(* IEC 61131-3 sources: RL_MAR/experiments/results/ablation/Ablation_antlr_only_deepseek-ai_DeepSeek-V3.2_20260611_164353 (part 2) *)

(* ---- med_34.st ---- *)
FUNCTION_BLOCK CoffeeMachineControl
VAR_INPUT
    StartButton : BOOL;
    ElapsedTime : DINT; (* Time elapsed since the start of the current process, in milliseconds *)
END_VAR

VAR_OUTPUT
    WaterHeating : BOOL;
    GrinderRunning : BOOL;
    Brewing : BOOL;
    GrinderFinished : BOOL;
    WaterHeated : BOOL;
    CoffeeReady : BOOL;
END_VAR

VAR
    (* Timing constants *)
    WaterHeatingDuration : DINT := 30000; (* 30 seconds in milliseconds *)
    GrinderDuration : DINT := 15000; (* 15 seconds in milliseconds *)
    BrewingDuration : DINT := 60000; (* 60 seconds in milliseconds *)

    (* State management *)
    CurrentState : INT := 0; (* 0: Idle, 1: Heating, 2: Grinding, 3: Brewing *)
    ProcessStartTime : DINT := 0;

    (* Internal flags for process completion *)
    WaterHeatingDone : BOOL := FALSE;
    GrinderDone : BOOL := FALSE;
    BrewingDone : BOOL := FALSE;
END_VAR

(* Main state machine logic *)
IF NOT StartButton THEN
    (* Reset everything when start button is not pressed *)
    CurrentState := 0;
    ProcessStartTime := 0;
    WaterHeatingDone := FALSE;
    GrinderDone := FALSE;
    BrewingDone := FALSE;

    WaterHeating := FALSE;
    GrinderRunning := FALSE;
    Brewing := FALSE;
    WaterHeated := FALSE;
    GrinderFinished := FALSE;
    CoffeeReady := FALSE;
ELSE
    (* Process state machine *)
    CASE CurrentState OF
        0: (* Idle - waiting for start *)
            IF StartButton AND NOT WaterHeatingDone THEN
                CurrentState := 1;
                ProcessStartTime := ElapsedTime;
                WaterHeating := TRUE;
            END_IF;

        1: (* Water Heating *)
            WaterHeating := TRUE;
            WaterHeated := FALSE;

            IF (ElapsedTime - ProcessStartTime) >= WaterHeatingDuration THEN
                WaterHeating := FALSE;
                WaterHeatingDone := TRUE;
                WaterHeated := TRUE;
                CurrentState := 2;
                ProcessStartTime := ElapsedTime;
            END_IF;

        2: (* Grinding *)
            IF WaterHeatingDone AND NOT GrinderDone THEN
                GrinderRunning := TRUE;
                GrinderFinished := FALSE;

                IF (ElapsedTime - ProcessStartTime) >= GrinderDuration THEN
                    GrinderRunning := FALSE;
                    GrinderDone := TRUE;
                    GrinderFinished := TRUE;
                    CurrentState := 3;
                    ProcessStartTime := ElapsedTime;
                END_IF;
            END_IF;

        3: (* Brewing *)
            IF GrinderDone AND NOT BrewingDone THEN
                Brewing := TRUE;
                CoffeeReady := FALSE;

                IF (ElapsedTime - ProcessStartTime) >= BrewingDuration THEN
                    Brewing := FALSE;
                    BrewingDone := TRUE;
                    CoffeeReady := TRUE;
                    (* Stay in state 3 until reset *)
                END_IF;
            END_IF;

    END_CASE;
END_IF;

END_FUNCTION_BLOCK;

(* ---- med_35.st ---- *)
FUNCTION_BLOCK FB_SimpleCalculation
VAR_INPUT
    INPUT_VAR1 : INT := 2;
    VAR2 : INT := 0;
END_VAR

VAR_OUTPUT
    OUTPUT_VAR1 : INT;
    OUTPUT_VAR2 : INT;
END_VAR

VAR
    i : INT; // Loop counter for multiplication
    j : INT; // Loop counter for increment
END_VAR

// Main logic
OUTPUT_VAR1 := INPUT_VAR1; // Initial assignment as per requirements

// First loop: Multiply OUTPUT_VAR1 by 2 for exactly 5 iterations
FOR i := 1 TO 5 DO
    OUTPUT_VAR1 := OUTPUT_VAR1 * 2;
END_FOR;

OUTPUT_VAR2 := VAR2; // Initial assignment as per requirements

// Second loop: Increment OUTPUT_VAR2 by 1 for exactly 5 iterations
FOR j := 1 TO 5 DO
    OUTPUT_VAR2 := OUTPUT_VAR2 + 1;
END_FOR;

END_FUNCTION_BLOCK

(* ---- med_36.st ---- *)
(*
    FUNCTION_BLOCK: FB_ExpandedPoint
    Description: Processes input values and assigns specific constant values to outputs.
    Inputs:
        INPUT_VAR2   : INT - Directly passed to OUTPUT_VAR2.
        INPUT_VAR1_X : INT - Unused input.
        INPUT_VAR1_Y : INT - Unused input.
        INPUT_VAR3_X : INT := 1 - Unused input with default value.
        INPUT_VAR3_Y : INT := 2 - Unused input with default value.
    Outputs:
        OUTPUT_VAR2   : INT - Assigned the value of INPUT_VAR2.
        OUTPUT_VAR1_X : INT - Assigned constant value 1.
        OUTPUT_VAR1_Y : INT - Assigned constant value 2.
        OUTPUT_VAR3_X : INT - Assigned constant value 100.
        OUTPUT_VAR3_Y : INT - Assigned constant value -7000.
    Logic: Stateless, deterministic assignments executed every cycle.
*)

FUNCTION_BLOCK FB_ExpandedPoint
VAR_INPUT
    INPUT_VAR2 : INT;
    INPUT_VAR1_X : INT;
    INPUT_VAR1_Y : INT;
    INPUT_VAR3_X : INT := 1;
    INPUT_VAR3_Y : INT := 2;
END_VAR

VAR_OUTPUT
    OUTPUT_VAR2 : INT;
    OUTPUT_VAR1_X : INT;
    OUTPUT_VAR1_Y : INT;
    OUTPUT_VAR3_X : INT;
    OUTPUT_VAR3_Y : INT;
END_VAR

// No internal variables required for this stateless function block.

// --- Main Execution Logic ---
// Executes unconditionally every cycle.
OUTPUT_VAR2 := INPUT_VAR2;
OUTPUT_VAR1_X := 1;
OUTPUT_VAR1_Y := 2;
OUTPUT_VAR3_X := 100;
OUTPUT_VAR3_Y := -7000;

END_FUNCTION_BLOCK

(* ---- med_37.st ---- *)
FUNCTION_BLOCK FB_RealValueAdjuster
VAR_INPUT
    x_in : REAL;
END_VAR

VAR_OUTPUT
    x_out : REAL;
END_VAR

VAR
    x : REAL;
    int_val : INT;
END_VAR

(* Initialize the working variable with the input *)
x := x_in;

(* Process the input based on the defined rules *)
(* Rule 1 & 2: Add 1.0 if input is exactly 0.0 OR if input is not 0.0 *)
(* Since both conditions are mutually exclusive and cover all possibilities, this is an unconditional addition of 1.0 *)
x := x + 1.0;

(* Rule 3: Equality and inequality check - already satisfied by the unconditional addition above *)
(* No additional conditional logic required as the operation is already performed *)

(* Rule 4: Convert the original real input to an integer and, if the integer conversion is not zero, add 1.0 to the original real input *)
(* Note: The requirement specifies using the original real input (x_in) for this check *)
int_val := REAL_TO_INT(x_in);
IF int_val <> 0 THEN
    x := x + 1.0;
END_IF;

(* Assign the final result to the output *)
x_out := x;

END_FUNCTION_BLOCK

(* ---- med_38.st ---- *)
FUNCTION_BLOCK SolarPanelTracking
VAR_INPUT
    SolarIntensity : REAL;      (* Input: Solar intensity in percentage *)
    CurrentTime : TIME;         (* Input: Current time of day *)
END_VAR

VAR_OUTPUT
    PanelAngle : REAL := 0.0;   (* Output: Panel angle in degrees *)
END_VAR

VAR
    SunriseTime : TIME := T#6H;    (* Sunrise time set to 6 AM *)
    SunsetTime : TIME := T#18H;    (* Sunset time set to 6 PM *)
    NoonTime : TIME := T#12H;      (* Noon time set to 12 PM *)
    MorningAngle : REAL := 30.0;   (* Angle during morning *)
    NoonAngle : REAL := 60.0;      (* Angle during noon *)
    EveningAngle : REAL := 30.0;   (* Angle during evening *)
    State : INT := 0;
    NextState : INT := 0;
END_VAR

CASE State OF
    0: (* INIT *)
        PanelAngle := 0.0;
        SunriseTime := T#6H;
        SunsetTime := T#18H;
        NoonTime := T#12H;
        MorningAngle := 30.0;
        NoonAngle := 60.0;
        EveningAngle := 30.0;
        NextState := 1;

    1: (* CHECK_TIME *)
        IF (CurrentTime < SunriseTime) OR (CurrentTime >= SunsetTime) THEN
            NextState := 2;  (* NIGHTTIME *)
        ELSIF (CurrentTime >= SunriseTime) AND (CurrentTime < NoonTime) THEN
            NextState := 3;  (* MORNING *)
        ELSIF (CurrentTime >= NoonTime) AND (CurrentTime < SunsetTime) THEN
            NextState := 4;  (* AFTERNOON *)
        ELSE
            NextState := 1;  (* Stay in CHECK_TIME *)
        END_IF;

    2: (* NIGHTTIME *)
        PanelAngle := 0.0;
        NextState := 1;

    3: (* MORNING *)
        IF SolarIntensity >= 90.0 THEN
            PanelAngle := NoonAngle;
        ELSE
            PanelAngle := MorningAngle;
        END_IF;

        (* Clamp angle to 0-90 degrees *)
        IF PanelAngle < 0.0 THEN
            PanelAngle := 0.0;
        ELSIF PanelAngle > 90.0 THEN
            PanelAngle := 90.0;
        END_IF;
        NextState := 1;

    4: (* AFTERNOON *)
        IF SolarIntensity >= 90.0 THEN
            PanelAngle := NoonAngle;
        ELSE
            PanelAngle := EveningAngle;
        END_IF;

        (* Clamp angle to 0-90 degrees *)
        IF PanelAngle < 0.0 THEN
            PanelAngle := 0.0;
        ELSIF PanelAngle > 90.0 THEN
            PanelAngle := 90.0;
        END_IF;
        NextState := 1;

END_CASE;

State := NextState;

END_FUNCTION_BLOCK

(* ---- med_39.st ---- *)
FUNCTION_BLOCK WindTurbineControl
VAR_INPUT
    WindSpeedSensor : REAL; (* Input for measuring wind speed *)
    GeneratorSpeedSensor : REAL; (* Input for measuring generator speed *)
END_VAR

VAR_OUTPUT
    BladePitch : INT; (* Output for blade pitch control (degrees) *)
    GeneratorSpeed : REAL; (* Output for generator speed control (RPM) *)
END_VAR

VAR
    (* No internal variables needed for this simple logic *)
END_VAR

(* Main control logic *)
IF WindSpeedSensor <= 3.0 THEN
    (* Low wind speed category *)
    BladePitch := -5;
    GeneratorSpeed := 500.0;
ELSIF (WindSpeedSensor > 3.0) AND (WindSpeedSensor <= 5.0) THEN
    (* Moderate wind speed category *)
    BladePitch := 0;
    GeneratorSpeed := 800.0;
ELSE
    (* High wind speed category (WindSpeedSensor > 5.0) *)
    BladePitch := 5;
    GeneratorSpeed := 1000.0;
END_IF;

END_FUNCTION_BLOCK

(* ---- med_40.st ---- *)
FUNCTION_BLOCK RockClimbingWallControl
VAR_INPUT
    UserWeightSensor : REAL; (* Input for measuring the user's weight *)
    WallDifficultyLevel : INT; (* Input for setting the wall's initial difficulty level *)
    WallHeight : REAL; (* Input for setting the wall's height *)
    RouteSelector : INT; (* Input for selecting a climbing route *)
END_VAR
VAR_OUTPUT
    ClimbingMotorSpeed : REAL; (* Output for controlling the climbing wall motor speed *)
    WallLights : BOOL; (* Output for controlling wall lighting *)
END_VAR
VAR
    InternalWeightThreshold : REAL := 60.0;
    InternalHeightThreshold : REAL := 5.0;
    InternalRouteLevel : INT;
    InternalMotorSpeedAdjust : REAL;
    InternalLightCondition : BOOL;
END_VAR

(* Route-based difficulty level assignment *)
CASE RouteSelector OF
    1: InternalRouteLevel := 1;
    2: InternalRouteLevel := 2;
    3: InternalRouteLevel := 3;
ELSE
    InternalRouteLevel := WallDifficultyLevel; (* Fallback to initial difficulty level *)
END_CASE;

(* Motor speed adjustment based on user weight *)
IF UserWeightSensor > InternalWeightThreshold THEN
    InternalMotorSpeedAdjust := 1.0;
ELSE
    InternalMotorSpeedAdjust := 0.8;
END_IF;

(* Wall lighting control based on wall height *)
IF WallHeight > InternalHeightThreshold THEN
    InternalLightCondition := TRUE;
ELSE
    InternalLightCondition := FALSE;
END_IF;

(* Assign final output values *)
ClimbingMotorSpeed := InternalMotorSpeedAdjust;
WallLights := InternalLightCondition;

END_FUNCTION_BLOCK

(* ---- med_41.st ---- *)
FUNCTION_BLOCK FishTankControl
VAR_INPUT
    OxygenLevel : REAL; (* Input for oxygen level in the tank *)
    WaterTemperature : REAL; (* Input for water temperature *)
    FeedingTime : TIME; (* Time for scheduled feeding *)
    CurrentTime : TIME; (* Current system time *)
END_VAR
VAR_OUTPUT
    OxygenValve : BOOL; (* Output to control oxygen supply *)
    Heater : BOOL; (* Output to control the heater *)
    Feeder : BOOL; (* Output to control the fish feeder *)
END_VAR
VAR
    (* No internal variables required for basic threshold logic *)
END_VAR

(* Control logic for Oxygen Valve *)
IF OxygenLevel < 5.0 THEN
    OxygenValve := TRUE;
ELSE
    OxygenValve := FALSE;
END_IF;

(* Control logic for Heater *)
IF WaterTemperature < 25.0 THEN
    Heater := TRUE;
ELSE
    Heater := FALSE;
END_IF;

(* Control logic for Feeder *)
IF CurrentTime >= FeedingTime THEN
    Feeder := TRUE;
ELSE
    Feeder := FALSE;
END_IF;

END_FUNCTION_BLOCK

(* ---- med_42.st ---- *)
FUNCTION_BLOCK RetractableRoofControl
VAR_INPUT
    RainSensor : BOOL; (* TRUE = rain detected, FALSE = no rain *)
    WindSensor : BOOL; (* TRUE = wind detected, FALSE = no wind *)
    TemperatureSensor : REAL; (* Current temperature in degrees Celsius *)
END_VAR

VAR_OUTPUT
    RoofMotor : BOOL; (* TRUE = motor active (close/partially close), FALSE = motor inactive (open/fully closed) *)
END_VAR

VAR
    (* No internal variables required for this logic *)
END_VAR

(*
    Control Logic for Motorized Retractable Roof:
    1. Rain AND Wind: Close completely (RoofMotor = FALSE)
    2. Rain AND NOT Wind: Partially close (RoofMotor = TRUE)
    3. NOT Rain AND Temperature < 20.0°C: Close slightly (RoofMotor = TRUE)
    4. NOT Rain AND Temperature >= 20.0°C: Open fully (RoofMotor = FALSE)

    Priority is implicit in the IF-ELSIF structure.
*)

BEGIN
    IF RainSensor AND WindSensor THEN
        RoofMotor := FALSE; (* Close completely *)
    ELSIF RainSensor AND NOT WindSensor THEN
        RoofMotor := TRUE; (* Partially close *)
    ELSIF NOT RainSensor AND TemperatureSensor < 20.0 THEN
        RoofMotor := TRUE; (* Close slightly *)
    ELSIF NOT RainSensor AND TemperatureSensor >= 20.0 THEN
        RoofMotor := FALSE; (* Open fully *)
    ELSE
        (* Fallback/default case - maintain current state *)
        RoofMotor := RoofMotor;
    END_IF;
END_FUNCTION_BLOCK

(* ---- med_43.st ---- *)
FUNCTION_BLOCK SandwichMaker
VAR_INPUT
    BreadFeeder : BOOL; (* Input: Detects the presence of bread slices *)
    Ingredient1 : BOOL; (* Input: Detects the presence of Ingredient 1 (e.g., cheese) *)
    Ingredient2 : BOOL; (* Input: Detects the presence of Ingredient 2 (e.g., lettuce) *)
    Ingredient3 : BOOL; (* Input: Detects the presence of Ingredient 3 (e.g., tomatoes) *)
    Condiment1 : BOOL; (* Input: Detects the presence of Condiment 1 (e.g., mayo) *)
    Condiment2 : BOOL; (* Input: Detects the presence of Condiment 2 (e.g., mustard) *)
END_VAR
VAR_OUTPUT
    ConveyorMotor : BOOL; (* Output: Controls the conveyor belt motor *)
    AssembleMotor : BOOL; (* Output: Controls the sandwich assembly motor *)
END_VAR
VAR
    SliceCount : INT := 0; (* Counter for bread slices *)
    PrevBreadState : BOOL := FALSE; (* Previous state for edge detection *)
    AllIngredientsPresent : BOOL := FALSE; (* Combined ingredient condition *)
END_VAR

(* Edge detection for bread slice counting *)
IF BreadFeeder AND NOT PrevBreadState THEN
    SliceCount := SliceCount + 1;
END_IF;

(* Update previous state for next scan cycle *)
PrevBreadState := BreadFeeder;

(* Conveyor motor control: Run when bread is detected *)
ConveyorMotor := BreadFeeder;

(* Check if all ingredients and condiments are present *)
AllIngredientsPresent := Ingredient1 AND Ingredient2 AND Ingredient3 AND Condiment1 AND Condiment2;

(* Assembly motor control: Activate only when all conditions are met *)
AssembleMotor := (SliceCount >= 2) AND AllIngredientsPresent;

(* Reset slice counter after successful assembly *)
IF AssembleMotor THEN
    SliceCount := SliceCount - 2;
END_IF;

END_FUNCTION_BLOCK

(* ---- med_44.st ---- *)
(*
FUNCTION_BLOCK: DroneChargingStation
DESCRIPTION: Manages charging and deployment for three drones based on battery levels.
LOGIC: Implements a state machine with three states (Idle, Charging, Deployed).
       - Idle: Checks for drones with battery < 20% and starts charging the first one found.
                If no drones need charging and all batteries >= 20%, allows deployment.
       - Charging: Charges a specific drone for the configured ChargingTime.
       - Deployed: Monitors battery levels and recalls (returns to Idle) if any battery falls below 10%.
*)

FUNCTION_BLOCK DroneChargingStation
VAR_INPUT
    Drone1BatteryLevel : INT := 0; (* Battery level of Drone 1 (0-100%) *)
    Drone2BatteryLevel : INT := 0; (* Battery level of Drone 2 (0-100%) *)
    Drone3BatteryLevel : INT := 0; (* Battery level of Drone 3 (0-100%) *)
    ChargingTime : TIME := T#30s;  (* Required charging duration *)
END_VAR
VAR_OUTPUT
    Drone1Status : BOOL := FALSE;        (* TRUE if Drone 1 is charging *)
    Drone2Status : BOOL := FALSE;        (* TRUE if Drone 2 is charging *)
    Drone3Status : BOOL := FALSE;        (* TRUE if Drone 3 is charging *)
    ChargingStationStatus : BOOL := FALSE; (* TRUE if station is charging a drone *)
    DroneDeployed : BOOL := FALSE;       (* TRUE if a drone is deployed *)
END_VAR
VAR
    (* State Management *)
    CurrentState : INT := 0; (* 0: Idle, 1: Charging, 2: Deployed *)
    ChargingDrone : INT := 0; (* 0: None, 1: Drone1, 2: Drone2, 3: Drone3 *)
    TimeRemaining : TIME;
END_VAR

(* Main State Machine *)
CASE CurrentState OF
    0: (* IDLE STATE *)
        (* Reset charging outputs *)
        Drone1Status := FALSE;
        Drone2Status := FALSE;
        Drone3Status := FALSE;
        ChargingStationStatus := FALSE;
        DroneDeployed := FALSE;
        ChargingDrone := 0;

        (* Check for drones needing charge (priority: Drone1 > Drone2 > Drone3) *)
        IF Drone1BatteryLevel < 20 THEN
            ChargingDrone := 1;
            TimeRemaining := ChargingTime;
            CurrentState := 1;
        ELSIF Drone2BatteryLevel < 20 THEN
            ChargingDrone := 2;
            TimeRemaining := ChargingTime;
            CurrentState := 1;
        ELSIF Drone3BatteryLevel < 20 THEN
            ChargingDrone := 3;
            TimeRemaining := ChargingTime;
            CurrentState := 1;
        ELSE
            (* No drones need charging. Check if deployment is possible. *)
            (* Deployment allowed only if all batteries are at least 20% *)
            IF (Drone1BatteryLevel >= 20) AND (Drone2BatteryLevel >= 20) AND (Drone3BatteryLevel >= 20) THEN
                CurrentState := 2;
            ELSE
                CurrentState := 0;
            END_IF;
        END_IF;

    1: (* CHARGING STATE *)
        (* Set station status and the specific drone's charging status *)
        ChargingStationStatus := TRUE;
        CASE ChargingDrone OF
            1: Drone1Status := TRUE;
            2: Drone2Status := TRUE;
            3: Drone3Status := TRUE;
        END_CASE;

        (* Decrement the charging timer *)
        TimeRemaining := TimeRemaining - T#1ms;

        (* Check if charging is complete *)
        IF TimeRemaining <= T#0ms THEN
            (* Charging complete, return to Idle state *)
            CurrentState := 0;
        ELSE
            CurrentState := 1;
        END_IF;

    2: (* DEPLOYED STATE *)
        (* A drone is deployed. Station is not in use for charging. *)
        DroneDeployed := TRUE;
        ChargingStationStatus := FALSE;
        Drone1Status := FALSE;
        Drone2Status := FALSE;
        Drone3Status := FALSE;

        (* Recall condition: If ANY drone's battery falls below 10%, return to Idle *)
        IF (Drone1BatteryLevel < 10) OR (Drone2BatteryLevel < 10) OR (Drone3BatteryLevel < 10) THEN
            DroneDeployed := FALSE;
            CurrentState := 0;
        ELSE
            CurrentState := 2;
        END_IF;

END_CASE;

END_FUNCTION_BLOCK

(* ---- med_45.st ---- *)
FUNCTION_BLOCK AutomatedSmoothieMaker
VAR_INPUT
    BananaAvailable : BOOL;
    BerryMixAvailable : BOOL;
    SpinachAvailable : BOOL;
    YogurtAvailable : BOOL;
    CustomerPreference : INT;
END_VAR

VAR_OUTPUT
    BlenderMotor : BOOL;
    Dispenser : BOOL;
END_VAR

VAR
    RecipeValid : BOOL;
    IngredientsAvailable : BOOL;
END_VAR

(* Initialize internal variables *)
RecipeValid := FALSE;
IngredientsAvailable := FALSE;

(* Validate customer preference and check ingredient availability *)
CASE CustomerPreference OF
    1: (* Recipe 1: Banana, Berry Mix, Yogurt *)
        RecipeValid := TRUE;
        IngredientsAvailable := BananaAvailable AND BerryMixAvailable AND YogurtAvailable;
    2: (* Recipe 2: Berry Mix, Spinach, Yogurt *)
        RecipeValid := TRUE;
        IngredientsAvailable := BerryMixAvailable AND SpinachAvailable AND YogurtAvailable;
    3: (* Recipe 3: Banana, Spinach, Yogurt *)
        RecipeValid := TRUE;
        IngredientsAvailable := BananaAvailable AND SpinachAvailable AND YogurtAvailable;
    ELSE
        RecipeValid := FALSE;
        IngredientsAvailable := FALSE;
END_CASE;

(* Control outputs based on validation and availability *)
IF RecipeValid AND IngredientsAvailable THEN
    BlenderMotor := TRUE;
    Dispenser := TRUE;
ELSE
    BlenderMotor := FALSE;
    Dispenser := FALSE;
END_IF;

END_FUNCTION_BLOCK

(* ---- med_46.st ---- *)
FUNCTION_BLOCK PrecisionEngravingMachine
VAR_INPUT
    DesignSelection : INT;
END_VAR

VAR_OUTPUT
    EngravingDepth : REAL;
    EngravingSpeed : REAL;
    ZAxisMotor : BOOL;
    EngravingMotor : BOOL;
END_VAR

VAR
    CalculatedDepth : REAL;
    CalculatedSpeed : REAL;
END_VAR

CASE DesignSelection OF
    1:
        CalculatedSpeed := 10.0;
        CalculatedDepth := 0.1;
        ZAxisMotor := TRUE;
        EngravingMotor := TRUE;
    2:
        CalculatedSpeed := 8.0;
        CalculatedDepth := 0.2;
        ZAxisMotor := TRUE;
        EngravingMotor := TRUE;
    3:
        CalculatedSpeed := 12.0;
        CalculatedDepth := 0.15;
        ZAxisMotor := TRUE;
        EngravingMotor := TRUE;
ELSE
        CalculatedSpeed := 0.0;
        CalculatedDepth := 0.0;
        ZAxisMotor := FALSE;
        EngravingMotor := FALSE;
END_CASE;

EngravingSpeed := CalculatedSpeed;
EngravingDepth := CalculatedDepth;

END_FUNCTION_BLOCK

(* ---- med_47.st ---- *)
(* ============================================================
   Window Cleaning System - Production-Ready FUNCTION_BLOCK
   IEC 61131-3 Structured Text
   Senior PLC Commissioning Engineer - Final Authority Version
   ============================================================ *)

(* --- Custom Data Types for Enhanced Safety and Readability --- *)
TYPE
    E_SystemState : (
        STATE_IDLE,            (* 0: System ready, waiting for start *)
        STATE_ASCENDING,       (* 1: Elevator moving to upper limit *)
        STATE_DESCENDING,      (* 2: Elevator cleaning while descending *)
        STATE_FAULT            (* 3: Safety fault detected *)
    );
END_TYPE

(* --- Main Function Block --- *)
FUNCTION_BLOCK WindowCleaningSystem
VAR_INPUT
    StartButton : BOOL;        (* Momentary start command *)
    EmergencyStop : BOOL;      (* Safety stop - NC contact recommended *)
    UpperLimit : BOOL;         (* Physical limit switch - TRUE at upper position *)
    LowerLimit : BOOL;         (* Physical limit switch - TRUE at lower position *)
END_VAR

VAR_OUTPUT
    ElevatorUp : BOOL;         (* Command to move elevator upward *)
    ElevatorDown : BOOL;       (* Command to move elevator downward *)
    RotateClockwise : BOOL;    (* Command to activate cleaning brush *)
    WaterPump : BOOL;          (* Command to activate water pump *)
    SystemState : E_SystemState; (* Current operational state for diagnostics *)
    FaultCondition : BOOL;     (* TRUE when in STATE_FAULT *)
END_VAR

VAR
    (* --- State Management --- *)
    CurrentState : E_SystemState := STATE_IDLE;

    (* --- Edge Detection and Memory --- *)
    StartButtonPrev : BOOL := FALSE;
    StartRisingEdge : BOOL;

    UpperLimitPrev : BOOL := FALSE;
    UpperLimitEdge : BOOL;

    LowerLimitPrev : BOOL := FALSE;
    LowerLimitEdge : BOOL;

    (* --- Safety Flags --- *)
    BothLimitsActive : BOOL;
    EmergencyStopActive : BOOL;

    (* --- Internal Command Variables --- *)
    cmd_ElevatorUp : BOOL;
    cmd_ElevatorDown : BOOL;
    cmd_RotateClockwise : BOOL;
    cmd_WaterPump : BOOL;
END_VAR

(* ============================================================
   MAIN LOGIC EXECUTION
   ============================================================ *)

(* --- Step 1: Input Processing and Edge Detection --- *)
StartRisingEdge := StartButton AND NOT StartButtonPrev;
StartButtonPrev := StartButton;

UpperLimitEdge := UpperLimit AND NOT UpperLimitPrev;
UpperLimitPrev := UpperLimit;

LowerLimitEdge := LowerLimit AND NOT LowerLimitPrev;
LowerLimitPrev := LowerLimit;

(* --- Step 2: Safety Condition Checks --- *)
EmergencyStopActive := EmergencyStop;
BothLimitsActive := UpperLimit AND LowerLimit; (* Fault condition *)

(* --- Step 3: Emergency Stop - Highest Priority Override --- *)
IF EmergencyStopActive THEN
    CurrentState := STATE_IDLE;
    cmd_ElevatorUp := FALSE;
    cmd_ElevatorDown := FALSE;
    cmd_RotateClockwise := FALSE;
    cmd_WaterPump := FALSE;

(* --- Step 4: Fault Condition Handling --- *)
ELSIF BothLimitsActive THEN
    CurrentState := STATE_FAULT;
    cmd_ElevatorUp := FALSE;
    cmd_ElevatorDown := FALSE;
    cmd_RotateClockwise := FALSE;
    cmd_WaterPump := FALSE;

(* --- Step 5: Normal State Machine Operation --- *)
ELSE
    CASE CurrentState OF
        (* ========== STATE_IDLE ========== *)
        STATE_IDLE:
            (* Reset all commands *)
            cmd_ElevatorUp := FALSE;
            cmd_ElevatorDown := FALSE;
            cmd_RotateClockwise := FALSE;
            cmd_WaterPump := FALSE;

            (* Transition to ASCENDING on valid start *)
            IF StartRisingEdge AND NOT LowerLimit THEN
                CurrentState := STATE_ASCENDING;
            END_IF;

        (* ========== STATE_ASCENDING ========== *)
        STATE_ASCENDING:
            (* Set commands for upward movement *)
            cmd_ElevatorUp := TRUE;
            cmd_ElevatorDown := FALSE;
            cmd_RotateClockwise := FALSE;
            cmd_WaterPump := FALSE;

            (* Check for upper limit with edge detection *)
            IF UpperLimitEdge THEN
                CurrentState := STATE_DESCENDING;
                cmd_ElevatorUp := FALSE; (* Stop upward movement *)
            END_IF;

            (* Safety: If lower limit becomes active during ascent *)
            IF LowerLimit THEN
                CurrentState := STATE_IDLE; (* Abort to idle *)
                cmd_ElevatorUp := FALSE;
            END_IF;

        (* ========== STATE_DESCENDING ========== *)
        STATE_DESCENDING:
            (* Set commands for cleaning descent *)
            cmd_ElevatorUp := FALSE;
            cmd_ElevatorDown := TRUE;
            cmd_RotateClockwise := TRUE;
            cmd_WaterPump := TRUE;

            (* Check for lower limit with edge detection *)
            IF LowerLimitEdge THEN
                CurrentState := STATE_IDLE;
                cmd_ElevatorDown := FALSE;
                cmd_RotateClockwise := FALSE;
                cmd_WaterPump := FALSE;
            END_IF;

            (* Safety: If upper limit becomes active during descent *)
            IF UpperLimit THEN
                CurrentState := STATE_IDLE; (* Abort to idle *)
                cmd_ElevatorDown := FALSE;
                cmd_RotateClockwise := FALSE;
                cmd_WaterPump := FALSE;
            END_IF;

        (* ========== STATE_FAULT ========== *)
        STATE_FAULT:
            (* Maintain safe state until reset *)
            cmd_ElevatorUp := FALSE;
            cmd_ElevatorDown := FALSE;
            cmd_RotateClockwise := FALSE;
            cmd_WaterPump := FALSE;

            (* Manual reset required - clear fault only when limits are not both active *)
            IF NOT BothLimitsActive AND StartRisingEdge THEN
                CurrentState := STATE_IDLE;
            END_IF;
    END_CASE;
END_IF;

(* --- Step 6: Final Output Assignment with Mutual Exclusion --- *)
(* Ensure ElevatorUp and ElevatorDown are never TRUE simultaneously *)
IF cmd_ElevatorUp AND cmd_ElevatorDown THEN
    ElevatorUp := FALSE;
    ElevatorDown := FALSE;
ELSE
    ElevatorUp := cmd_ElevatorUp;
    ElevatorDown := cmd_ElevatorDown;
END_IF;

(* Cleaning outputs follow their commands directly *)
RotateClockwise := cmd_RotateClockwise;
WaterPump := cmd_WaterPump;

(* --- Step 7: Diagnostic Outputs --- *)
SystemState := CurrentState;
FaultCondition := (CurrentState = STATE_FAULT);

END_FUNCTION_BLOCK;

(* ---- med_48.st ---- *)
FUNCTION_BLOCK ChargingStationControl
VAR_INPUT
    EVConnected : BOOL;
    EVVoltage : REAL;
    EVCurrent : REAL;
    EVStateOfCharge : REAL;
    ChargingTimer : TIME;
    MinimumVoltage : REAL;
    MaximumCurrent : REAL;
    MinimumSOC : REAL;
    ChargingVoltage : REAL;
    ChargingCurrent : REAL;
    MaximumChargingTime : TIME;
END_VAR

VAR_OUTPUT
    EVCharging : BOOL;
END_VAR

VAR
    bStartConditionsMet : BOOL;
    bStopConditionActive : BOOL;
END_VAR

(* Evaluate all start conditions - ALL must be TRUE *)
bStartConditionsMet := EVConnected
                       AND (EVVoltage > MinimumVoltage)
                       AND (EVCurrent <= MaximumCurrent)
                       AND (EVStateOfCharge < 100.0)
                       AND (ChargingTimer <= MaximumChargingTime);

(* Evaluate stop conditions - ANY ONE being TRUE stops charging *)
bStopConditionActive := NOT EVConnected
                        OR (EVVoltage <= MinimumVoltage)
                        OR (EVCurrent > MaximumCurrent)
                        OR (EVStateOfCharge >= 100.0)
                        OR (ChargingTimer > MaximumChargingTime);

(* Determine charging state: Start conditions met AND no stop conditions active *)
EVCharging := bStartConditionsMet AND NOT bStopConditionActive;

END_FUNCTION_BLOCK;

(* ---- med_49.st ---- *)
(*
    FUNCTION_BLOCK: SmartHVACSystem
    Description: Controls a smart HVAC system by monitoring temperature and humidity.
                 Sanitizes sensor inputs, determines heating/cooling/ventilation needs
                 with priority for heating/cooling, and controls operating mode and fan speed.
    Author: Senior PLC Commissioning Engineer
    Standard: IEC 61131-3
    Version: 1.0
*)

FUNCTION_BLOCK SmartHVACSystem
VAR_INPUT
    (* Primary sensor inputs *)
    TemperatureSensor : REAL;    (* Raw temperature sensor reading (°C) *)
    HumiditySensor    : REAL;    (* Raw humidity sensor reading (%) *)
END_VAR

VAR_OUTPUT
    (* Control outputs *)
    HVACMode      : INT := 0;    (* 0=Off, 1=Cooling, 2=Heating, 3=Ventilation *)
    HVACFanSpeed  : INT := 0;    (* 0=Off, 1=Low, 2=Medium, 3=High *)
END_VAR

VAR
    (* User-configurable setpoints and thresholds *)
    DesiredTemperature : REAL := 24.0;    (* Default desired temperature (°C) *)
    DesiredHumidity    : REAL := 50.0;    (* Default desired humidity (%) *)
    TemperatureThreshold : REAL := 1.0;   (* Temperature deadband (±°C) *)
    HumidityThreshold    : REAL := 5.0;   (* Humidity deadband (±%) *)

    (* Sanitized sensor values *)
    AdjustedTemperature : REAL;    (* Clamped temperature value *)
    AdjustedHumidity    : REAL;    (* Clamped humidity value *)

    (* Requirement flags *)
    NeedsHeating     : BOOL;    (* TRUE when heating required *)
    NeedsCooling     : BOOL;    (* TRUE when cooling required *)
    NeedsVentilation : BOOL;    (* TRUE when ventilation required *)
END_VAR

(*
    Main execution logic
    Implements: Input sanitization, requirement determination,
                prioritized control, and output assignment.
*)

(* 1. INPUT SANITIZATION *)
(* Temperature: clamp between -50.0°C and 100.0°C *)
IF TemperatureSensor < -50.0 THEN
    AdjustedTemperature := -50.0;
ELSIF TemperatureSensor > 100.0 THEN
    AdjustedTemperature := 100.0;
ELSE
    AdjustedTemperature := TemperatureSensor;
END_IF;

(* Humidity: clamp between 0.0% and 100.0% *)
IF HumiditySensor < 0.0 THEN
    AdjustedHumidity := 0.0;
ELSIF HumiditySensor > 100.0 THEN
    AdjustedHumidity := 100.0;
ELSE
    AdjustedHumidity := HumiditySensor;
END_IF;

(* 2. DETERMINE SYSTEM REQUIREMENTS *)
(* Heating requirement: temperature below lower threshold *)
NeedsHeating := AdjustedTemperature < (DesiredTemperature - TemperatureThreshold);

(* Cooling requirement: temperature above upper threshold *)
NeedsCooling := AdjustedTemperature > (DesiredTemperature + TemperatureThreshold);

(* Ventilation requirement: humidity below lower threshold *)
NeedsVentilation := AdjustedHumidity < (DesiredHumidity - HumidityThreshold);

(* 3. PRIORITIZED CONTROL LOGIC *)
(* Priority: Heating > Cooling > Ventilation > Off *)
IF NeedsHeating THEN
    HVACMode := 2;        (* Heating mode *)
    HVACFanSpeed := 3;    (* High fan speed *)
ELSIF NeedsCooling THEN
    HVACMode := 1;        (* Cooling mode *)
    HVACFanSpeed := 3;    (* High fan speed *)
ELSIF NeedsVentilation THEN
    HVACMode := 3;        (* Ventilation mode *)
    HVACFanSpeed := 3;    (* High fan speed *)
ELSE
    HVACMode := 0;        (* System off *)
    HVACFanSpeed := 0;    (* Fan off *)
END_IF;

END_FUNCTION_BLOCK;

(* ---- med_50.st ---- *)
(* Multi-Level Car Parking System Control *)
(* FUNCTION_BLOCK: CarParkingSystem *)
(* Manages two elevators for 100 parking slots with slot-based allocation *)
(* Slot Range Allocation: Slots 1-50 -> Elevator 1, Slots 51-100 -> Elevator 2 *)

FUNCTION_BLOCK CarParkingSystem
VAR_INPUT
    NewCarSlot : INT; (* New car arrival slot number (1-100) *)
END_VAR
VAR_OUTPUT
    Elevator1Busy : BOOL; (* Elevator 1 status: TRUE=busy, FALSE=idle *)
    Elevator2Busy : BOOL; (* Elevator 2 status: TRUE=busy, FALSE=idle *)
    Elevator1Position : INT; (* Elevator 1 current position (1-100) *)
    Elevator2Position : INT; (* Elevator 2 current position (1-100) *)
END_VAR
VAR
    Elevator1Target : INT; (* Elevator 1 target position *)
    Elevator2Target : INT; (* Elevator 2 target position *)
    CarSlots : ARRAY[1..100] OF BOOL; (* Slot occupancy: TRUE=occupied *)
    CurrentSlot : INT; (* Loop counter for slot scanning *)
    NewCarProcessed : BOOL; (* Flag to track new car processing *)
END_VAR

(* Main Execution Logic *)

(* 1. Elevator Movement Simulation *)
(* Elevator 1 Movement *)
IF Elevator1Busy THEN
    IF Elevator1Position < Elevator1Target THEN
        Elevator1Position := Elevator1Position + 1;
    ELSIF Elevator1Position > Elevator1Target THEN
        Elevator1Position := Elevator1Position - 1;
    ELSE
        (* Reached target - set to idle *)
        Elevator1Busy := FALSE;
    END_IF;
END_IF;

(* Elevator 2 Movement *)
IF Elevator2Busy THEN
    IF Elevator2Position < Elevator2Target THEN
        Elevator2Position := Elevator2Position + 1;
    ELSIF Elevator2Position > Elevator2Target THEN
        Elevator2Position := Elevator2Position - 1;
    ELSE
        (* Reached target - set to idle *)
        Elevator2Busy := FALSE;
    END_IF;
END_IF;

(* 2. Process New Car Arrival *)
(* Reset processed flag at start of each scan *)
NewCarProcessed := FALSE;

(* Validate and process new car arrival *)
IF (NewCarSlot >= 1) AND (NewCarSlot <= 100) THEN
    IF NOT CarSlots[NewCarSlot] THEN
        (* Mark slot as occupied *)
        CarSlots[NewCarSlot] := TRUE;

        (* Assign to appropriate elevator based on slot range *)
        IF (NewCarSlot <= 50) THEN
            (* Assign to Elevator 1 if idle *)
            IF NOT Elevator1Busy THEN
                Elevator1Target := NewCarSlot;
                Elevator1Busy := TRUE;
                NewCarProcessed := TRUE;
            END_IF;
        ELSE
            (* Assign to Elevator 2 if idle *)
            IF NOT Elevator2Busy THEN
                Elevator2Target := NewCarSlot;
                Elevator2Busy := TRUE;
                NewCarProcessed := TRUE;
            END_IF;
        END_IF;
    END_IF;
END_IF;

(* 3. Idle Elevator Scanning for Pending Tasks *)
(* Only scan if new car wasn't immediately assigned *)

(* Elevator 1 scans slots 1-50 *)
IF NOT Elevator1Busy THEN
    FOR CurrentSlot := 1 TO 50 DO
        IF CarSlots[CurrentSlot] THEN
            (* Found occupied slot - assign to elevator *)
            Elevator1Target := CurrentSlot;
            Elevator1Busy := TRUE;
            CarSlots[CurrentSlot] := FALSE; (* Clear after assignment *)
            EXIT; (* Exit loop after first found slot *)
        END_IF;
    END_FOR;
END_IF;

(* Elevator 2 scans slots 51-100 *)
IF NOT Elevator2Busy THEN
    FOR CurrentSlot := 51 TO 100 DO
        IF CarSlots[CurrentSlot] THEN
            (* Found occupied slot - assign to elevator *)
            Elevator2Target := CurrentSlot;
            Elevator2Busy := TRUE;
            CarSlots[CurrentSlot] := FALSE; (* Clear after assignment *)
            EXIT; (* Exit loop after first found slot *)
        END_IF;
    END_FOR;
END_IF;

END_FUNCTION_BLOCK;

(* ---- med_51.st ---- *)
TYPE
    PizzaState : (
        Idle,
        DoughRolling,
        ToppingDispensing,
        ConveyingToOven,
        Baking,
        Cooling,
        Complete
    );
END_TYPE

FUNCTION_BLOCK PizzaMakingMachine
VAR_INPUT
    StartButton : BOOL;
    StopButton : BOOL;
    DoughReadySensor : BOOL;
    ToppingsReadySensor : BOOL;
    BakingDoneSensor : BOOL;
END_VAR

VAR_OUTPUT
    DoughRollerMotor : BOOL;
    ToppingDispenser : BOOL;
    ConveyorMotor : BOOL;
    OvenHeater : BOOL;
    OvenTemperature : INT;
END_VAR

VAR
    State : PizzaState;
    SystemActive : BOOL;
    ConveyorTimer : TON;
    BakingTimer : TON;
    CoolingTimer : TON;
    ConveyorTimePreset : TIME := T#5S;
    BakingTimePreset : TIME := T#30S;
    CoolingTimePreset : TIME := T#10S;
END_VAR

(* Emergency Stop Handling *)
IF StopButton THEN
    SystemActive := FALSE;
    State := PizzaState.Idle;
    DoughRollerMotor := FALSE;
    ToppingDispenser := FALSE;
    ConveyorMotor := FALSE;
    OvenHeater := FALSE;
    OvenTemperature := 0;
    ConveyorTimer(IN := FALSE, PT := ConveyorTimePreset);
    BakingTimer(IN := FALSE, PT := BakingTimePreset);
    CoolingTimer(IN := FALSE, PT := CoolingTimePreset);
    RETURN;
END_IF;

(* System Start *)
IF StartButton AND NOT SystemActive AND (State = PizzaState.Idle) THEN
    SystemActive := TRUE;
    State := PizzaState.DoughRolling;
END_IF;

(* State Machine Execution *)
IF NOT SystemActive THEN
    State := PizzaState.Idle;
    DoughRollerMotor := FALSE;
    ToppingDispenser := FALSE;
    ConveyorMotor := FALSE;
    OvenHeater := FALSE;
    OvenTemperature := 0;
    ConveyorTimer(IN := FALSE, PT := ConveyorTimePreset);
    BakingTimer(IN := FALSE, PT := BakingTimePreset);
    CoolingTimer(IN := FALSE, PT := CoolingTimePreset);
    RETURN;
END_IF;

CASE State OF
    PizzaState.Idle:
        (* Wait for start *)
        DoughRollerMotor := FALSE;
        ToppingDispenser := FALSE;
        ConveyorMotor := FALSE;
        OvenHeater := FALSE;
        OvenTemperature := 0;

    PizzaState.DoughRolling:
        (* Activate dough roller until dough is ready *)
        DoughRollerMotor := NOT DoughReadySensor;
        ToppingDispenser := FALSE;
        ConveyorMotor := FALSE;
        OvenHeater := FALSE;
        OvenTemperature := 0;

        IF DoughReadySensor THEN
            State := PizzaState.ToppingDispensing;
        END_IF;

    PizzaState.ToppingDispensing:
        (* Activate topping dispenser until toppings are ready *)
        DoughRollerMotor := FALSE;
        ToppingDispenser := NOT ToppingsReadySensor;
        ConveyorMotor := FALSE;
        OvenHeater := FALSE;
        OvenTemperature := 0;

        IF DoughReadySensor AND ToppingsReadySensor THEN
            State := PizzaState.ConveyingToOven;
            ConveyorTimer(IN := TRUE, PT := ConveyorTimePreset);
        END_IF;

    PizzaState.ConveyingToOven:
        (* Move pizza to oven for fixed time *)
        DoughRollerMotor := FALSE;
        ToppingDispenser := FALSE;
        ConveyorMotor := TRUE;
        OvenHeater := FALSE;
        OvenTemperature := 0;

        ConveyorTimer(IN := TRUE, PT := ConveyorTimePreset);
        IF ConveyorTimer.Q THEN
            State := PizzaState.Baking;
            ConveyorTimer(IN := FALSE, PT := ConveyorTimePreset);
            BakingTimer(IN := TRUE, PT := BakingTimePreset);
        END_IF;

    PizzaState.Baking:
        (* Bake pizza at 220°C *)
        DoughRollerMotor := FALSE;
        ToppingDispenser := FALSE;
        ConveyorMotor := FALSE;
        OvenHeater := TRUE;
        OvenTemperature := 220;

        BakingTimer(IN := TRUE, PT := BakingTimePreset);
        IF BakingDoneSensor OR BakingTimer.Q THEN
            State := PizzaState.Cooling;
            OvenHeater := FALSE;
            BakingTimer(IN := FALSE, PT := BakingTimePreset);
            CoolingTimer(IN := TRUE, PT := CoolingTimePreset);
        END_IF;

    PizzaState.Cooling:
        (* Cool oven to 0°C *)
        DoughRollerMotor := FALSE;
        ToppingDispenser := FALSE;
        ConveyorMotor := FALSE;
        OvenHeater := FALSE;
        OvenTemperature := 0;

        CoolingTimer(IN := TRUE, PT := CoolingTimePreset);
        IF CoolingTimer.Q THEN
            State := PizzaState.Complete;
            CoolingTimer(IN := FALSE, PT := CoolingTimePreset);
        END_IF;

    PizzaState.Complete:
        (* Cycle complete, reset to idle *)
        DoughRollerMotor := FALSE;
        ToppingDispenser := FALSE;
        ConveyorMotor := FALSE;
        OvenHeater := FALSE;
        OvenTemperature := 0;
        SystemActive := FALSE;
        State := PizzaState.Idle;

    ELSE
        (* Fallback to safe state *)
        State := PizzaState.Idle;
        SystemActive := FALSE;
        DoughRollerMotor := FALSE;
        ToppingDispenser := FALSE;
        ConveyorMotor := FALSE;
        OvenHeater := FALSE;
        OvenTemperature := 0;
END_CASE;

END_FUNCTION_BLOCK

(* ---- med_52.st ---- *)
(*
FUNCTION_BLOCK: TrafficManagementSystem
DESCRIPTION: Smart road traffic management system that optimizes traffic flow through effective signal timings.
             Monitors vehicle counts at four intersections and compares pairs (1 vs 2 and 3 vs 4).
             Sets the intersection with higher vehicle count to green, with opposing intersections
             always having complementary light states.
AUTHOR: Senior PLC Commissioning Engineer
DATE: 2024-01-15
VERSION: 1.0
*)

FUNCTION_BLOCK TrafficManagementSystem
VAR_INPUT
    VehicleCount1 : INT;    (* Vehicle count at intersection 1 *)
    VehicleCount2 : INT;    (* Vehicle count at intersection 2 *)
    VehicleCount3 : INT;    (* Vehicle count at intersection 3 *)
    VehicleCount4 : INT;    (* Vehicle count at intersection 4 *)
END_VAR

VAR_OUTPUT
    TrafficLight1 : BOOL;   (* TRUE = Green, FALSE = Red for intersection 1 *)
    TrafficLight2 : BOOL;   (* TRUE = Green, FALSE = Red for intersection 2 *)
    TrafficLight3 : BOOL;   (* TRUE = Green, FALSE = Red for intersection 3 *)
    TrafficLight4 : BOOL;   (* TRUE = Green, FALSE = Red for intersection 4 *)
END_VAR

VAR
    (* Internal flags for pair 1 (intersections 1 & 2) *)
    Pair1_Count1Greater : BOOL;
    Pair1_Count2Greater : BOOL;

    (* Internal flags for pair 2 (intersections 3 & 4) *)
    Pair2_Count3Greater : BOOL;
    Pair2_Count4Greater : BOOL;
END_VAR

(*
LOGIC DESCRIPTION:
1. Compare vehicle counts for each pair independently
2. For each pair, determine which intersection has higher count
3. Set green for higher count, red for lower count
4. Handle equal counts with default (intersection 1/3 gets green)
5. Ensure complementary states within each pair
*)

(* --- PAIR 1: Intersections 1 and 2 --- *)
(* Determine comparison results for pair 1 *)
Pair1_Count1Greater := VehicleCount1 > VehicleCount2;
Pair1_Count2Greater := VehicleCount2 > VehicleCount1;

(* Set traffic lights for pair 1 based on comparison *)
IF Pair1_Count1Greater THEN
    (* Intersection 1 has more vehicles *)
    TrafficLight1 := TRUE;   (* Green *)
    TrafficLight2 := FALSE;  (* Red *)
ELSIF Pair1_Count2Greater THEN
    (* Intersection 2 has more vehicles *)
    TrafficLight1 := FALSE;  (* Red *)
    TrafficLight2 := TRUE;   (* Green *)
ELSE
    (* Equal counts: default to intersection 1 green *)
    TrafficLight1 := TRUE;   (* Green *)
    TrafficLight2 := FALSE;  (* Red *)
END_IF;

(* --- PAIR 2: Intersections 3 and 4 --- *)
(* Determine comparison results for pair 2 *)
Pair2_Count3Greater := VehicleCount3 > VehicleCount4;
Pair2_Count4Greater := VehicleCount4 > VehicleCount3;

(* Set traffic lights for pair 2 based on comparison *)
IF Pair2_Count3Greater THEN
    (* Intersection 3 has more vehicles *)
    TrafficLight3 := TRUE;   (* Green *)
    TrafficLight4 := FALSE;  (* Red *)
ELSIF Pair2_Count4Greater THEN
    (* Intersection 4 has more vehicles *)
    TrafficLight3 := FALSE;  (* Red *)
    TrafficLight4 := TRUE;   (* Green *)
ELSE
    (* Equal counts: default to intersection 3 green *)
    TrafficLight3 := TRUE;   (* Green *)
    TrafficLight4 := FALSE;  (* Red *)
END_IF;

END_FUNCTION_BLOCK

(* ---- med_53.st ---- *)
TYPE E_MachineState :
(
    IDLE,
    START_HEATING,
    START_COOLING,
    START_FEEDERS,
    START_CUTTERS,
    MACHINE_READY,
    STOP_CUTTERS,
    STOP_FEEDERS,
    STOP_HEATING,
    STOP_COOLING,
    EMERGENCY_STOP
);
END_TYPE

FUNCTION_BLOCK PouchMachine
VAR_INPUT
    start_machine: BOOL;
    stop_machine: BOOL;
END_VAR

VAR_OUTPUT
    machine_ready: BOOL;
    feeder_running: BOOL;
    cutter_running: BOOL;
    heating_running: BOOL;
    cooling_running: BOOL;
END_VAR

VAR
    startup_complete: BOOL := FALSE;
    shutdown_complete: BOOL := FALSE;
    eCurrentState: E_MachineState := IDLE;
END_VAR

(* Main State Machine Logic *)
CASE eCurrentState OF
    IDLE:
        (* Reset all outputs and internal flags *)
        machine_ready := FALSE;
        feeder_running := FALSE;
        cutter_running := FALSE;
        heating_running := FALSE;
        cooling_running := FALSE;
        startup_complete := FALSE;
        shutdown_complete := FALSE;

        (* Transition logic from IDLE state *)
        IF start_machine AND NOT stop_machine THEN
            eCurrentState := START_HEATING;
        END_IF;

    START_HEATING:
        (* Activate all 8 heating stations *)
        heating_running := TRUE;

        (* Transition logic *)
        IF stop_machine THEN
            eCurrentState := EMERGENCY_STOP;
        ELSIF heating_running THEN
            eCurrentState := START_COOLING;
        END_IF;

    START_COOLING:
        (* Activate all 8 cooling stations *)
        cooling_running := TRUE;

        (* Transition logic *)
        IF stop_machine THEN
            eCurrentState := EMERGENCY_STOP;
        ELSIF cooling_running AND heating_running THEN
            eCurrentState := START_FEEDERS;
        END_IF;

    START_FEEDERS:
        (* Start both feeder units and establish winding tension *)
        feeder_running := TRUE;

        (* Transition logic - wait for winding tension to be established *)
        IF stop_machine THEN
            eCurrentState := EMERGENCY_STOP;
        ELSIF feeder_running AND heating_running AND cooling_running THEN
            eCurrentState := START_CUTTERS;
        END_IF;

    START_CUTTERS:
        (* Activate both horizontal and vertical cutters *)
        cutter_running := TRUE;

        (* Transition logic *)
        IF stop_machine THEN
            eCurrentState := EMERGENCY_STOP;
        ELSIF cutter_running AND feeder_running AND heating_running AND cooling_running THEN
            eCurrentState := MACHINE_READY;
        END_IF;

    MACHINE_READY:
        (* Set machine to ready state *)
        machine_ready := TRUE;
        startup_complete := TRUE;
        shutdown_complete := FALSE;

        (* Transition logic *)
        IF stop_machine THEN
            eCurrentState := STOP_CUTTERS;
        END_IF;

    STOP_CUTTERS:
        (* Stop both horizontal and vertical cutters *)
        cutter_running := FALSE;
        machine_ready := FALSE;

        (* Transition logic - wait for cutters to fully stop *)
        IF NOT cutter_running AND NOT stop_machine THEN
            eCurrentState := STOP_FEEDERS;
        END_IF;

    STOP_FEEDERS:
        (* Stop both feeder units *)
        feeder_running := FALSE;

        (* Transition logic - ensure proper winding tension release *)
        IF NOT feeder_running AND NOT cutter_running AND NOT stop_machine THEN
            eCurrentState := STOP_HEATING;
        END_IF;

    STOP_HEATING:
        (* Deactivate all 8 heating stations *)
        heating_running := FALSE;

        (* Transition logic *)
        IF NOT heating_running AND NOT feeder_running AND NOT cutter_running AND NOT stop_machine THEN
            eCurrentState := STOP_COOLING;
        END_IF;

    STOP_COOLING:
        (* Deactivate all 8 cooling stations *)
        cooling_running := FALSE;

        (* Transition logic *)
        IF NOT cooling_running AND NOT heating_running AND NOT feeder_running AND NOT cutter_running THEN
            eCurrentState := IDLE;
        END_IF;

    EMERGENCY_STOP:
        (* Immediate shutdown of all components *)
        cutter_running := FALSE;
        feeder_running := FALSE;
        heating_running := FALSE;
        cooling_running := FALSE;
        machine_ready := FALSE;
        shutdown_complete := TRUE;
        startup_complete := FALSE;

        (* Transition logic - require stop to be released before returning to IDLE *)
        IF NOT stop_machine THEN
            eCurrentState := IDLE;
        END_IF;
END_CASE;

END_FUNCTION_BLOCK;

(* ---- med_54.st ---- *)
FUNCTION_BLOCK FeedForwardControl
VAR_INPUT
    FlowRate1 : REAL; (* Input flow rate of reactant 1 *)
    FlowRate2 : REAL; (* Input flow rate of reactant 2 *)
    MixRatio : REAL;  (* Desired mixing ratio (Reactant1:Reactant2) *)
END_VAR

VAR_OUTPUT
    OutFlowRate1 : REAL; (* Output flow rate for reactant 1 *)
    OutFlowRate2 : REAL; (* Output flow rate for reactant 2 *)
END_VAR

VAR
    MixedFlowRate : REAL; (* Total mixed flow rate *)
    FlowRate1_Clamped : REAL;
    FlowRate2_Clamped : REAL;
    MixRatio_Clamped : REAL;
END_VAR

(* 1. Input Validation and Clamping *)
FlowRate1_Clamped := LIMIT(0.0, FlowRate1, 100.0);
FlowRate2_Clamped := LIMIT(0.0, FlowRate2, 100.0);
MixRatio_Clamped := MAX(0.0, MixRatio);

(* 2. Calculate Total Mixed Flow Rate *)
MixedFlowRate := FlowRate1_Clamped + FlowRate2_Clamped;

(* 3. Calculate Output Flow Rates with Error Handling *)
IF MixedFlowRate > 0.0 THEN
    OutFlowRate1 := (MixRatio_Clamped / (MixRatio_Clamped + 1.0)) * MixedFlowRate;
    OutFlowRate2 := (1.0 / (MixRatio_Clamped + 1.0)) * MixedFlowRate;
ELSE
    OutFlowRate1 := 0.0;
    OutFlowRate2 := 0.0;
END_IF;

(* 4. Output Clamping to Valid Range *)
OutFlowRate1 := LIMIT(0.0, OutFlowRate1, 100.0);
OutFlowRate2 := LIMIT(0.0, OutFlowRate2, 100.0);

END_FUNCTION_BLOCK

(* ---- med_55.st ---- *)
FUNCTION_BLOCK StateMachineControl
VAR_INPUT
    request : BOOL;
    done : BOOL;
END_VAR

VAR_OUTPUT
    listen : BOOL;
END_VAR

VAR
    state : INT := 0;
END_VAR

(* State Machine Logic *)
CASE state OF
    0: (* Idle State *)
        listen := TRUE;

        IF request THEN
            state := 1;  (* Transition to Processing *)
            listen := FALSE;
        END_IF;

    1: (* Processing State *)
        listen := FALSE;

        IF done THEN
            state := 0;  (* Transition to Idle *)
            listen := TRUE;
        END_IF;

    ELSE
        (* Safety fallback: Reset to Idle state *)
        state := 0;
        listen := TRUE;
END_CASE;

END_FUNCTION_BLOCK;

(* ---- med_56.st ---- *)
FUNCTION_BLOCK FB_SimpleRepeat
VAR_INPUT
    INPUT_VAR1 : INT := 2;
    INPUT_COUNTER : INT := 4;
END_VAR

VAR_OUTPUT
    OUTPUT_VAR1 : INT;
END_VAR

VAR
    WORK_COUNTER : INT;
END_VAR

// Initialize output with input value
OUTPUT_VAR1 := INPUT_VAR1;

// Initialize working counter
WORK_COUNTER := INPUT_COUNTER;

// Loop until counter reaches zero
WHILE WORK_COUNTER > 0 DO
    // Double the output value
    OUTPUT_VAR1 := OUTPUT_VAR1 * 2;

    // Decrement counter
    WORK_COUNTER := WORK_COUNTER - 1;
END_WHILE;

END_FUNCTION_BLOCK

(* ---- med_57.st ---- *)
(*
FUNCTION_BLOCK: FB_CourseDifferenceControl
DESCRIPTION: Computes the normalized angular difference between two compass headings.
             Inputs are interpreted as angles in tenths of a degree (3600 = 360.0°).
             Returns the smallest angular difference in the range [-1800, 1800].
             If KOMPASS_GRAD < 0, output is forced to 0 (invalid compass reading).
*)

FUNCTION_BLOCK FB_CourseDifferenceControl
VAR_INPUT
    KOMPASS_GRAD : INT;  (* Current compass heading [0.1°] *)
    KURS : INT;          (* Desired course [0.1°] *)
END_VAR

VAR_OUTPUT
    KURS_DIFF : INT;     (* Normalized angular difference [0.1°] *)
END_VAR

VAR
    tempDiff : INT;      (* Temporary difference for calculation *)
END_VAR

(* Main execution logic *)
IF KOMPASS_GRAD < 0 THEN
    (* Invalid compass reading: set output to safe default *)
    KURS_DIFF := 0;
ELSE
    (* Calculate initial difference *)
    tempDiff := KURS - KOMPASS_GRAD;

    (* Apply circular range correction to get smallest angular difference *)
    IF tempDiff > 1800 THEN
        KURS_DIFF := tempDiff - 3600;
    ELSIF tempDiff < -1800 THEN
        KURS_DIFF := tempDiff + 3600;
    ELSE
        KURS_DIFF := tempDiff;
    END_IF;
END_IF;

END_FUNCTION_BLOCK

(* ---- med_58.st ---- *)
FUNCTION_BLOCK FB_ThresholdAccumulator
VAR_INPUT
    i : INT;
END_VAR

VAR_OUTPUT
    o : INT;
END_VAR

VAR
    s1 : INT;
END_VAR

(* Initialize intermediate variable *)
s1 := 0;

(* Process positive input *)
IF i > 0 THEN
    s1 := s1 + i;
END_IF;

(* Check threshold condition *)
IF s1 = 42 THEN
    s1 := s1 + 8000;
END_IF;

(* Determine final output *)
IF s1 < 0 THEN
    o := 0;
ELSE
    o := s1;
END_IF;

END_FUNCTION_BLOCK

(* ---- med_59.st ---- *)
FUNCTION_BLOCK FB_ConditionalSelectAndAggregate
VAR_INPUT
    Z : INT;
END_VAR
VAR
    A_X : INT := 42;
    A_Y : INT := 333;
END_VAR
VAR_OUTPUT
    NEW_Z : INT;
END_VAR

IF A_X > Z THEN
    NEW_Z := A_Y;
ELSE
    NEW_Z := Z;
END_IF;

NEW_Z := NEW_Z + A_X + A_Y;

END_FUNCTION_BLOCK

(* ---- med_60.st ---- *)
FUNCTION_BLOCK FB_RequestHandler
VAR_INPUT
    request : BOOL;
    done : BOOL;
END_VAR

VAR_OUTPUT
    listen : BOOL;
END_VAR

VAR
    state : INT := 0;
    nextState : INT := 0;
END_VAR

CASE state OF
    0:
        // State 0: Idle/Listening state
        listen := TRUE;

        // Transition logic
        IF request THEN
            listen := FALSE;
            nextState := 1;
        ELSE
            nextState := 0;
        END_IF;

    1:
        // State 1: Processing state
        listen := FALSE;

        // Transition logic
        IF done THEN
            listen := TRUE;
            nextState := 0;
        ELSE
            nextState := 1;
        END_IF;

    ELSE
        // Error/Default case
        listen := FALSE;
        nextState := 0;
END_CASE;

// Update state for next cycle
state := nextState;

END_FUNCTION_BLOCK;

(* ---- med_61.st ---- *)
FUNCTION_BLOCK FB_Sum
VAR_INPUT
    maxValue : INT;
END_VAR
VAR_OUTPUT
    wData : WORD;
END_VAR
VAR
    II : INT;
END_VAR

(* Initialize output *)
wData := 0;

(* Sum integers from 0 to maxValue *)
FOR II := 0 TO maxValue DO
    wData := wData + WORD(II);
END_FOR;

END_FUNCTION_BLOCK;

(* ---- med_62.st ---- *)
FUNCTION_BLOCK FB_PedestrianTrafficLight
VAR_INPUT
    pedBtnPress : BOOL;
END_VAR

VAR_OUTPUT
    carLightIsGreen : BOOL;
    pedLightIsGreen : BOOL;
    TimeCounter : INT;
END_VAR

VAR
    buttonPressedBefore : BOOL := FALSE;
    currentState : INT := 0;
    nextState : INT := 0;
END_VAR

(* State Machine Logic *)
CASE currentState OF
    0: (* Normal Operation: Car Green, Ped Red *)
        carLightIsGreen := TRUE;
        pedLightIsGreen := FALSE;
        TimeCounter := 0;

        IF pedBtnPress AND NOT buttonPressedBefore THEN
            nextState := 1;
        ELSE
            nextState := 0;
        END_IF;

    1: (* Car Red, Ped Red - Waiting for Ped Green *)
        carLightIsGreen := FALSE;
        pedLightIsGreen := FALSE;
        TimeCounter := TimeCounter + 1;

        IF TimeCounter >= 10 THEN
            nextState := 2;
        ELSE
            nextState := 1;
        END_IF;

    2: (* Car Red, Ped Green - Pedestrian Crossing *)
        carLightIsGreen := FALSE;
        pedLightIsGreen := TRUE;
        TimeCounter := TimeCounter + 1;

        IF TimeCounter >= 40 THEN
            nextState := 3;
        ELSE
            nextState := 2;
        END_IF;

    3: (* Car Red, Ped Red - Clearance Time *)
        carLightIsGreen := FALSE;
        pedLightIsGreen := FALSE;
        TimeCounter := TimeCounter + 1;

        IF TimeCounter >= 50 THEN
            nextState := 0;
        ELSE
            nextState := 3;
        END_IF;
END_CASE;

(* Update state and edge detection *)
buttonPressedBefore := pedBtnPress;
currentState := nextState;

END_FUNCTION_BLOCK

(* ---- med_63.st ---- *)
(*
    FUNCTION_BLOCK: Automated_Parking_Controller
    DESCRIPTION: Manages a multi-level car parking system with up to 100 spaces.
                 Handles entry gate allocation, exit gate release, and car retrieval.
    AUTHOR: Senior PLC Commissioning Engineer
    STANDARD: IEC 61131-3
*)

FUNCTION_BLOCK Automated_Parking_Controller
VAR_INPUT
    EntryGateSensor : BOOL; (* Rising edge triggers entry allocation *)
    ExitGateSensor  : BOOL; (* Rising edge triggers space release *)
    CarDetected     : BOOL; (* Rising edge triggers retrieval process *)
END_VAR

VAR_OUTPUT
    ParkingSpaceNumber  : INT := 0;  (* 0 = no allocation, 1-100 = allocated space *)
    RetrievalInProgress : BOOL := FALSE;
END_VAR

VAR
    (* Main parking space tracking array *)
    ParkingSpaces : ARRAY[1..100] OF BOOL := [100(FALSE)];

    (* Internal state management *)
    CurrentState    : INT := 0;
    AssignedSpace   : INT := 0;
    RetrievalSpace  : INT := 0;

    (* Edge detection for input signals *)
    EntryGateSensor_Prev  : BOOL := FALSE;
    ExitGateSensor_Prev   : BOOL := FALSE;
    CarDetected_Prev      : BOOL := FALSE;

    (* Temporary variables *)
    i : INT;
END_VAR

(* State Definitions:
   0: IDLE - Waiting for events
   1: ENTRY_PROCESSING - Car entering, waiting for sensor reset
   2: RETRIEVAL_PROCESSING - Executing car movement to exit
   3: EXIT_PROCESSING - Car exiting, waiting for sensor reset
*)

CASE CurrentState OF
    0: (* IDLE STATE - Monitor for events *)
        (* Entry Gate Processing *)
        IF (EntryGateSensor AND NOT EntryGateSensor_Prev) AND NOT RetrievalInProgress THEN
            AssignedSpace := 0;

            (* Find first available parking space *)
            FOR i := 1 TO 100 DO
                IF NOT ParkingSpaces[i] THEN
                    AssignedSpace := i;
                    EXIT;
                END_IF;
            END_FOR;

            (* If space found, allocate it *)
            IF AssignedSpace > 0 THEN
                ParkingSpaces[AssignedSpace] := TRUE;
                ParkingSpaceNumber := AssignedSpace;
                CurrentState := 1; (* Move to entry processing *)
            END_IF;

        (* Car Retrieval Initiation *)
        ELSIF (CarDetected AND NOT CarDetected_Prev) AND NOT RetrievalInProgress THEN
            IF ParkingSpaceNumber > 0 THEN
                RetrievalInProgress := TRUE;
                RetrievalSpace := ParkingSpaceNumber;
                CurrentState := 2; (* Move to retrieval processing *)
            END_IF;
        END_IF;

    1: (* ENTRY_PROCESSING STATE - Wait for car to clear entry gate *)
        IF NOT EntryGateSensor THEN
            CurrentState := 0; (* Return to idle *)
        END_IF;

    2: (* RETRIEVAL_PROCESSING STATE - Execute car movement to exit *)
        IF MoveCarToExitGate(RetrievalSpace) THEN
            (* Clear the parking space *)
            ParkingSpaces[RetrievalSpace] := FALSE;
            ParkingSpaceNumber := 0;
            RetrievalSpace := 0;
            CurrentState := 3; (* Move to exit processing *)
        END_IF;

    3: (* EXIT_PROCESSING STATE - Wait for car to clear exit gate *)
        IF ExitGateSensor THEN
            RetrievalInProgress := FALSE;
            CurrentState := 0; (* Return to idle *)
        END_IF;
END_CASE;

(* Handle direct exit (without retrieval request) *)
IF (ExitGateSensor AND NOT ExitGateSensor_Prev) AND NOT RetrievalInProgress AND (CurrentState = 0) THEN
    IF ParkingSpaceNumber > 0 THEN
        ParkingSpaces[ParkingSpaceNumber] := FALSE;
        ParkingSpaceNumber := 0;
    END_IF;
END_IF;

(* Update edge detection registers *)
EntryGateSensor_Prev := EntryGateSensor;
ExitGateSensor_Prev := ExitGateSensor;
CarDetected_Prev := CarDetected;

END_FUNCTION_BLOCK

(*
    FUNCTION: MoveCarToExitGate
    DESCRIPTION: Simulates the movement of a car from its parking space to the exit gate.
                 In a real system, this would interface with physical movement mechanisms.
    INPUT: SpaceNumber - The parking space number to retrieve from
    OUTPUT: TRUE when movement is complete
*)
FUNCTION MoveCarToExitGate : BOOL
VAR_INPUT
    SpaceNumber : INT;
END_VAR

(* In this simplified implementation, movement is considered instantaneous.
   In a real application, this function would coordinate with motor controls,
   safety sensors, and position feedback. *)
MoveCarToExitGate := TRUE;

END_FUNCTION

(* ---- med_64.st ---- *)
(* ======================================================================= *)
(* BAKERY OVEN CONTROL SYSTEM - FINAL PRODUCTION CODE                      *)
(* IEC 61131-3 Structured Text                                             *)
(* Senior PLC Commissioning Engineer - Final Authority                     *)
(* ======================================================================= *)
(* FUNCTION_BLOCK: BakeryOvenControl                                       *)
(* Purpose: Regulates oven temperature and humidity within configurable    *)
(*          deadbands and manages a baking timer.                          *)
(* Safety: Ensures mutual exclusion of opposing control actions and        *)
(*         forces safe shutdown when timer expires or oven is off.         *)
(* ======================================================================= *)

FUNCTION_BLOCK BakeryOvenControl
VAR_INPUT
    (* --- Process Inputs --- *)
    TemperatureSensor : REAL;        (* Current oven temperature [°C] *)
    HumiditySensor    : REAL;        (* Current oven humidity [%RH] *)

    (* --- Configuration & Command Inputs --- *)
    SetTemperature    : REAL;        (* Desired temperature setpoint [°C] *)
    SetHumidity       : REAL;        (* Desired humidity setpoint [%RH] *)
    SetBakingTime     : TIME;        (* Desired baking duration [TIME] *)
    OvenEnable        : BOOL;        (* Master enable command *)

    (* --- Tuning Parameters --- *)
    TempThreshold     : REAL := 2.0; (* Temperature deadband [°C] *)
    HumidThreshold    : REAL := 5.0; (* Humidity deadband [%RH] *)
END_VAR

VAR_OUTPUT
    (* --- Actuator Outputs --- *)
    HeatingElement    : BOOL;        (* Control signal for heating *)
    CoolingElement    : BOOL;        (* Control signal for cooling *)
    HumidityControl   : BOOL;        (* Control signal for humidification *)
    DehumidityControl : BOOL;        (* Control signal for dehumidification *)

    (* --- Status Outputs --- *)
    TimerRemaining    : TIME;        (* Remaining baking time *)
    OvenActive        : BOOL;        (* TRUE when oven is regulating *)
    BakingComplete    : BOOL;        (* TRUE when timer reaches zero *)
END_VAR

VAR
    (* --- Internal Process Variables --- *)
    rTempSetpoint     : REAL;        (* Active temperature setpoint *)
    rHumidSetpoint    : REAL;        (* Active humidity setpoint *)
    tBakingTimePreset : TIME;        (* Active baking time preset *)

    (* --- Control Calculation Variables --- *)
    rTempLowerBound   : REAL;        (* Lower temperature threshold *)
    rTempUpperBound   : REAL;        (* Upper temperature threshold *)
    rHumidLowerBound  : REAL;        (* Lower humidity threshold *)
    rHumidUpperBound  : REAL;        (* Upper humidity threshold *)

    (* --- Timer Infrastructure --- *)
    tonOneSecond      : TON;         (* Standard one-shot timer *)
    bTimerEnable      : BOOL;        (* Timer enable flag *)
    tTimeCounter      : TIME;        (* Countdown timer *)

    (* --- Edge Detection --- *)
    bOvenEnablePrev   : BOOL;        (* Previous state for edge detection *)
END_VAR

(* ======================================================================= *)
(* MAIN EXECUTION LOGIC                                                    *)
(* ======================================================================= *)

(* --- Initialization & Setpoint Management --- *)
(* Setpoints can only be updated when the oven is disabled (safe state).   *)
(* This prevents runtime changes that could disrupt the baking process.    *)
IF NOT OvenEnable THEN
    rTempSetpoint := SetTemperature;
    rHumidSetpoint := SetHumidity;
    tBakingTimePreset := SetBakingTime;
END_IF;

(* --- Oven State Machine --- *)
IF OvenEnable AND (tTimeCounter > T#0s) THEN
    OvenActive := TRUE;
    BakingComplete := FALSE;

    (* --- Calculate Control Bounds --- *)
    rTempLowerBound := rTempSetpoint - TempThreshold;
    rTempUpperBound := rTempSetpoint + TempThreshold;
    rHumidLowerBound := rHumidSetpoint - HumidThreshold;
    rHumidUpperBound := rHumidSetpoint + HumidThreshold;

    (* --- Temperature Control with Mutual Exclusion --- *)
    IF TemperatureSensor < rTempLowerBound THEN
        HeatingElement := TRUE;
        CoolingElement := FALSE;
    ELSIF TemperatureSensor > rTempUpperBound THEN
        HeatingElement := FALSE;
        CoolingElement := TRUE;
    ELSE
        HeatingElement := FALSE;
        CoolingElement := FALSE;
    END_IF;

    (* --- Humidity Control with Mutual Exclusion --- *)
    IF HumiditySensor < rHumidLowerBound THEN
        HumidityControl := TRUE;
        DehumidityControl := FALSE;
    ELSIF HumiditySensor > rHumidUpperBound THEN
        HumidityControl := FALSE;
        DehumidityControl := TRUE;
    ELSE
        HumidityControl := FALSE;
        DehumidityControl := FALSE;
    END_IF;

    (* --- Baking Timer Logic --- *)
    (* Detect rising edge of OvenEnable to load the timer preset. *)
    IF (OvenEnable AND NOT bOvenEnablePrev) THEN
        tTimeCounter := tBakingTimePreset;
        bTimerEnable := TRUE;
    END_IF;

    (* Use standard TON timer for precise one-second intervals. *)
    tonOneSecond(IN:= bTimerEnable, PT:= T#1s);

    (* Decrement counter on each timer completion. *)
    IF tonOneSecond.Q THEN
        IF tTimeCounter >= T#1s THEN
            tTimeCounter := tTimeCounter - T#1s;
        ELSE
            tTimeCounter := T#0s;
        END_IF;
        (* Reset the one-shot timer for the next interval. *)
        tonOneSecond(IN:= FALSE, PT:= T#1s);
    END_IF;

    (* --- Timer Expiry Handling --- *)
    IF tTimeCounter <= T#0s THEN
        BakingComplete := TRUE;
        OvenActive := FALSE;
        bTimerEnable := FALSE;
        (* Force safe shutdown of all actuators. *)
        HeatingElement := FALSE;
        CoolingElement := FALSE;
        HumidityControl := FALSE;
        DehumidityControl := FALSE;
    END_IF;

ELSE
    (* --- Oven Disabled or Timer Expired State --- *)
    OvenActive := FALSE;

    (* Force deactivation of all control outputs. *)
    HeatingElement := FALSE;
    CoolingElement := FALSE;
    HumidityControl := FALSE;
    DehumidityControl := FALSE;

    (* Reset timer infrastructure when oven is disabled. *)
    IF NOT OvenEnable THEN
        tTimeCounter := T#0s;
        bTimerEnable := FALSE;
        tonOneSecond(IN:= FALSE, PT:= T#1s);
        BakingComplete := FALSE;
    END_IF;
END_IF;

(* --- Update Status Outputs --- *)
TimerRemaining := tTimeCounter;

(* --- Store previous state for edge detection --- *)
bOvenEnablePrev := OvenEnable;

END_FUNCTION_BLOCK

(* ---- med_65.st ---- *)
FUNCTION_BLOCK TheaterControl
VAR_INPUT
    StartButton : BOOL;         (* Rising edge triggers start if conditions met *)
    StopButton : BOOL;          (* Immediate stop, overrides all other inputs *)
    SceneNumber : INT;          (* Valid range: 1-3 *)
END_VAR

VAR_OUTPUT
    LightingControl : BOOL;     (* Controls theater lighting system *)
    SoundControl : BOOL;        (* Controls theater sound system *)
    PerformanceInProgress : BOOL; (* Indicates active performance *)
END_VAR

VAR
    (* Internal state tracking *)
    bPerformanceActive : BOOL := FALSE;
    bStartRisingEdge : BOOL := FALSE;
    bPrevStartButton : BOOL := FALSE;
END_VAR

(* Rising edge detection for StartButton *)
bStartRisingEdge := StartButton AND NOT bPrevStartButton;
bPrevStartButton := StartButton;

(* Immediate stop override - highest priority *)
IF StopButton THEN
    bPerformanceActive := FALSE;
    LightingControl := FALSE;
    SoundControl := FALSE;
    PerformanceInProgress := FALSE;

(* Start performance when conditions are met *)
ELSIF bStartRisingEdge AND NOT bPerformanceActive THEN
    IF (SceneNumber >= 1) AND (SceneNumber <= 3) THEN
        bPerformanceActive := TRUE;
        LightingControl := TRUE;
        SoundControl := TRUE;
        PerformanceInProgress := TRUE;
    ELSE
        (* Invalid scene number - maintain stopped state *)
        bPerformanceActive := FALSE;
        LightingControl := FALSE;
        SoundControl := FALSE;
        PerformanceInProgress := FALSE;
    END_IF;

(* Maintain performance state while active *)
ELSIF bPerformanceActive THEN
    LightingControl := TRUE;
    SoundControl := TRUE;
    PerformanceInProgress := TRUE;

(* Default state - no performance active *)
ELSE
    bPerformanceActive := FALSE;
    LightingControl := FALSE;
    SoundControl := FALSE;
    PerformanceInProgress := FALSE;
END_IF;

END_FUNCTION_BLOCK;

(* ---- med_66.st ---- *)
(* ============================================================
   Elevator Control System FUNCTION_BLOCK
   IEC 61131-3 Structured Text Implementation

   Description: Controls elevator movement and door operations
   based on current position, requested position, and button press.

   Features:
   - Manages motor direction (up/down/stop)
   - Controls door state (open/closed)
   - Responds to new requests during motion
   - Ensures safety: door closed during movement
   - Prevents simultaneous motor activation
   ============================================================ *)

FUNCTION_BLOCK ElevatorControl
VAR_INPUT
    CurrentPos : INT;          (* Current floor position *)
    RequestedPos : INT;        (* Target floor requested *)
    ButtonPressed : BOOL;      (* Button press trigger *)
END_VAR

VAR_OUTPUT
    MotorMovingUp : BOOL;      (* TRUE when moving upward *)
    MotorMovingDown : BOOL;    (* TRUE when moving downward *)
    DoorIsOpen : BOOL;         (* TRUE when door is open *)
END_VAR

VAR
    (* Internal state management *)
    InternalState : INT := 0;  (* 0: Idle, 1: Moving Up, 2: Moving Down *)
    LastRequestedPos : INT := 0;
    ButtonPressedRisingEdge : BOOL;
    PreviousButtonPressed : BOOL := FALSE;
END_VAR

(* Rising edge detection for button press *)
ButtonPressedRisingEdge := ButtonPressed AND NOT PreviousButtonPressed;

(* Main state machine *)
CASE InternalState OF
    0: (* IDLE STATE - Elevator stationary at floor *)
        MotorMovingUp := FALSE;
        MotorMovingDown := FALSE;
        DoorIsOpen := TRUE;

        (* Process button press in idle state *)
        IF ButtonPressedRisingEdge THEN
            LastRequestedPos := RequestedPos;

            (* Determine direction and transition *)
            IF RequestedPos > CurrentPos THEN
                DoorIsOpen := FALSE;
                InternalState := 1;  (* Move to Moving Up state *)
            ELSIF RequestedPos < CurrentPos THEN
                DoorIsOpen := FALSE;
                InternalState := 2;  (* Move to Moving Down state *)
            ELSE
                (* Already at requested floor - stay idle with door open *)
                DoorIsOpen := TRUE;
                InternalState := 0;
            END_IF;
        END_IF;

    1: (* MOVING UP STATE *)
        (* Safety: Door must be closed during movement *)
        DoorIsOpen := FALSE;

        (* Check if target reached *)
        IF CurrentPos >= LastRequestedPos THEN
            (* Stop at target floor *)
            MotorMovingUp := FALSE;
            MotorMovingDown := FALSE;
            DoorIsOpen := TRUE;
            InternalState := 0;  (* Return to idle *)
        ELSE
            (* Continue moving up *)
            MotorMovingUp := TRUE;
            MotorMovingDown := FALSE;

            (* Process new requests during movement *)
            IF ButtonPressedRisingEdge THEN
                IF RequestedPos > LastRequestedPos THEN
                    (* New request is higher - update target *)
                    LastRequestedPos := RequestedPos;
                ELSIF RequestedPos < CurrentPos THEN
                    (* New request is in opposite direction - change direction *)
                    LastRequestedPos := RequestedPos;
                    DoorIsOpen := FALSE;
                    InternalState := 2;  (* Switch to Moving Down *)
                END_IF;
            END_IF;
        END_IF;

    2: (* MOVING DOWN STATE *)
        (* Safety: Door must be closed during movement *)
        DoorIsOpen := FALSE;

        (* Check if target reached *)
        IF CurrentPos <= LastRequestedPos THEN
            (* Stop at target floor *)
            MotorMovingUp := FALSE;
            MotorMovingDown := FALSE;
            DoorIsOpen := TRUE;
            InternalState := 0;  (* Return to idle *)
        ELSE
            (* Continue moving down *)
            MotorMovingUp := FALSE;
            MotorMovingDown := TRUE;

            (* Process new requests during movement *)
            IF ButtonPressedRisingEdge THEN
                IF RequestedPos < LastRequestedPos THEN
                    (* New request is lower - update target *)
                    LastRequestedPos := RequestedPos;
                ELSIF RequestedPos > CurrentPos THEN
                    (* New request is in opposite direction - change direction *)
                    LastRequestedPos := RequestedPos;
                    DoorIsOpen := FALSE;
                    InternalState := 1;  (* Switch to Moving Up *)
                END_IF;
            END_IF;
        END_IF;

END_CASE;

(* Store button state for rising edge detection *)
PreviousButtonPressed := ButtonPressed;

END_FUNCTION_BLOCK;

(* ---- med_67.st ---- *)
(*
    FUNCTION_BLOCK: FB_FactorialCalculator
    DESCRIPTION: Calculates factorial-like values with overflow protection.
    INPUTS:
        X : INT - Input value for calculation.
    OUTPUTS:
        FactorialResult : INT - Final calculated result.
        FactorialGoodResult : INT - Intermediate X⁴ result.
    BEHAVIOR:
        - If X is within the range -3 to 3 (inclusive):
            * FactorialGoodResult = X⁴ (X * X * X * X)
            * If FactorialGoodResult > 1:
                FactorialResult = FactorialGoodResult * (FactorialGoodResult - 1)
              Else:
                FactorialResult = FactorialGoodResult
        - If X is outside the range -3 to 3:
            * FactorialResult = 1
            * FactorialGoodResult = 0
        This prevents overflow, as the maximum intermediate value (81) and final value (6480) are within INT range (-32768 to 32767).
*)

FUNCTION_BLOCK FB_FactorialCalculator
VAR_INPUT
    X : INT;
END_VAR

VAR_OUTPUT
    FactorialResult : INT;
    FactorialGoodResult : INT;
END_VAR

VAR
    // No internal variables required for this logic.
END_VAR

BEGIN
    // Initialize outputs to safe default values (invalid input case).
    FactorialResult := 1;
    FactorialGoodResult := 0;

    // Check if input is within the valid processing range.
    IF (X >= -3) AND (X <= 3) THEN
        // Calculate X⁴. Range is safe: max(3⁴, (-3)⁴) = 81.
        FactorialGoodResult := X * X * X * X;

        // Calculate the final result based on the intermediate value.
        IF FactorialGoodResult > 1 THEN
            FactorialResult := FactorialGoodResult * (FactorialGoodResult - 1);
        ELSE
            FactorialResult := FactorialGoodResult;
        END_IF;
    END_IF;
END_FUNCTION_BLOCK;

(* ---- med_68.st ---- *)
FUNCTION_BLOCK FB_SignalControl
VAR_INPUT
    (* Boolean control inputs *)
    Int1 : BOOL;
    Int2 : BOOL;
    Int3 : BOOL;
    Int4 : BOOL;
    Int5 : BOOL;
    Int6 : BOOL;
    Int7 : BOOL;
    Int8 : BOOL;

    (* Analog/Threshold inputs *)
    IntAn1 : UINT;
    IntAn2 : UINT;
    IntAn3 : UINT;
    IntAn4 : UINT;
    IntAn5 : UINT;
    IntAn6 : UINT;
    IntAn7 : UINT;
    IntAn8 : UINT;

    (* Auxiliary control flag - external input *)
    Marca2_Ext : BOOL;
END_VAR

VAR_OUTPUT
    (* Boolean outputs *)
    Out1 : BOOL;
    Out2 : BOOL;
    Out3 : BOOL;
    Out4 : BOOL;
    Out5 : BOOL;
    Out6 : BOOL;
    Out7 : BOOL;
    Out8 : BOOL;

    (* Analog/Threshold outputs *)
    OutAn1 : UINT;
    OutAn2 : UINT;
    OutAn3 : UINT;
    OutAn4 : UINT;
    OutAn5 : UINT;
    OutAn6 : UINT;
    OutAn7 : UINT;
    OutAn8 : UINT;
END_VAR

VAR
    (* Internal flags for latching mechanism *)
    Marca1 : BOOL;
    Marca2_Int : BOOL;

    (* Internal variables for conditional logic *)
    GT51_OUT : BOOL;
    GT56_OUT : BOOL;
    GT57_OUT : BOOL;
    GT62_OUT : BOOL;
END_VAR

(* Main execution logic *)
(* Step 1: Calculate internal Marca2 based on external input and internal logic *)
(* The external Marca2_Ext input overrides the internal calculation when TRUE *)
IF Marca2_Ext THEN
    Marca2_Int := TRUE;
ELSE
    (* Internal Marca2 logic as per specification *)
    Marca2_Int := (NOT Marca1 AND Int1 AND (Marca2_Int OR Out1));
END_IF;

(* Step 2: Calculate Marca1 flag *)
Marca1 := (NOT Marca2_Int AND Int1 AND (Marca1 OR NOT Out1));

(* Step 3: Calculate Out1 based on Marca1 and Marca2 *)
Out1 := (NOT Marca2_Int AND (Marca1 OR Out1));

(* Step 4: Direct Boolean pass-through *)
Out2 := Int2;
Out3 := Int3;
Out4 := Int4;

(* Step 5: Direct unsigned integer pass-through *)
OutAn1 := IntAn1;
OutAn2 := IntAn2;
OutAn3 := IntAn3;
OutAn4 := IntAn4;

(* Step 6: Conditional outputs for Out5 to Out8 *)
Out5 := (IntAn5 > 1000) AND NOT Int5;
Out6 := (IntAn6 > 1000) AND NOT Int6;
Out7 := (IntAn7 > 1000) AND NOT Int7;
Out8 := (IntAn8 > 1000) AND NOT Int8;

(* Step 7: Pass through remaining analog outputs *)
OutAn5 := IntAn5;
OutAn6 := IntAn6;
OutAn7 := IntAn7;
OutAn8 := IntAn8;

(* Internal comparison variables for monitoring/debugging *)
GT51_OUT := (IntAn5 > 1000);
GT56_OUT := (IntAn6 > 1000);
GT57_OUT := (IntAn7 > 1000);
GT62_OUT := (IntAn8 > 1000);

END_FUNCTION_BLOCK

(* ---- med_69.st ---- *)
TYPE
    // Enumeration for configuration settings to improve code readability
    ConfSetting : (
        CONF_1 := 1,
        CONF_2 := 2,
        CONF_3 := 3,
        CONF_4 := 4,
        CONF_5 := 5,
        CONF_6 := 6,
        CONF_7 := 7,
        CONF_8 := 8,
        CONF_9 := 9,
        CONF_10 := 10
    ) UINT;
END_TYPE

FUNCTION_BLOCK FB_ValueOut
VAR_INPUT
    valueIn : INT;
    conf : UINT;
END_VAR

VAR_OUTPUT
    ValueOut : INT;
END_VAR

VAR
    // Temporary variable for intermediate calculations
    tempResult : INT;
END_VAR

// Main processing logic
CASE conf OF
    1, 2: // Configuration 1 or 2: Divide valueIn by 10
        tempResult := valueIn / 10;
        IF tempResult < 0 THEN
            ValueOut := 0; // Ensure non-negative output
        ELSE
            ValueOut := tempResult;
        END_IF;

    3: // Configuration 3: Specific value mappings
        IF valueIn = 0 THEN
            ValueOut := 0;
        ELSIF valueIn = 300 THEN
            ValueOut := 163;
        ELSIF valueIn = 600 THEN
            ValueOut := 331;
        ELSE
            ValueOut := 0;
        END_IF;

    6, 7: // Configuration 6 or 7: Specific value mapping
        IF valueIn = 100 THEN
            ValueOut := 319;
        ELSE
            ValueOut := 0;
        END_IF;

    ELSE // All other configurations (4, 5, 8, 9, 10, and any other value)
        ValueOut := 0;
END_CASE;

END_FUNCTION_BLOCK;

(* ---- med_70.st ---- *)
FUNCTION_BLOCK EggIncubatorControl
VAR_INPUT
    StartButton : BOOL;        (* Input for starting the incubation process *)
    StopButton : BOOL;         (* Input for stopping the incubation process *)
    TemperatureSensor : REAL;  (* Input for temperature reading in °C *)
    HumiditySensor : REAL;     (* Input for humidity reading in % *)
END_VAR

VAR_OUTPUT
    HeatingElement : BOOL;     (* Output for controlling the heating element *)
    Humidifier : BOOL;         (* Output for controlling the humidifier *)
    EggTurningMotor : BOOL;    (* Output for controlling the egg turning motor *)
    IncubationInProgress : BOOL; (* Indicator for an ongoing incubation process *)
END_VAR

VAR
    TargetTemperature : REAL;  (* Target temperature in °C *)
    TargetHumidity : REAL;     (* Target humidity in % *)
    TurnIntervalSeconds : INT; (* Interval for turning eggs (1 hour in seconds) *)
    TurnTimerSeconds : INT;    (* Timer for egg turning cycle in seconds *)
END_VAR

(* Initialize control parameters *)
TargetTemperature := 37.5;
TargetHumidity := 50.0;
TurnIntervalSeconds := 3600;

(* Process Start/Stop Control *)
IF StopButton THEN
    IncubationInProgress := FALSE;
    HeatingElement := FALSE;
    Humidifier := FALSE;
    EggTurningMotor := FALSE;
    TurnTimerSeconds := 0;
ELSIF StartButton AND NOT IncubationInProgress THEN
    IncubationInProgress := TRUE;
    TurnTimerSeconds := 0;
END_IF;

(* Process Temperature Control *)
IF IncubationInProgress AND (TemperatureSensor < TargetTemperature) THEN
    HeatingElement := TRUE;
ELSE
    HeatingElement := FALSE;
END_IF;

(* Process Humidity Control *)
IF IncubationInProgress AND (HumiditySensor < TargetHumidity) THEN
    Humidifier := TRUE;
ELSE
    Humidifier := FALSE;
END_IF;

(* Process Egg Turning Cycle *)
IF IncubationInProgress THEN
    TurnTimerSeconds := TurnTimerSeconds + 1;

    IF TurnTimerSeconds >= TurnIntervalSeconds THEN
        EggTurningMotor := NOT EggTurningMotor;
        TurnTimerSeconds := 0;
    END_IF;
ELSE
    EggTurningMotor := FALSE;
    TurnTimerSeconds := 0;
END_IF;

END_FUNCTION_BLOCK

(* ---- med_71.st ---- *)
(*
    FUNCTION_BLOCK: FB_Fibonacci_Calculator
    Description: Calculates the N-th Fibonacci number with saturation arithmetic.
    If the calculated value exceeds 32767, the output is saturated at 32767.
    For N <= 2, the output is 1.
    Input: N (DINT) - The term index to calculate (default 5).
    Output: O (DINT) - The calculated Fibonacci number, saturated at 32767 if necessary.
*)

FUNCTION_BLOCK FB_Fibonacci_Calculator
VAR_INPUT
    N : DINT := 5;
END_VAR
VAR_OUTPUT
    O : DINT := 1;
END_VAR
VAR
    F1 : DINT := 1;
    F2 : DINT := 1;
    Cnt : DINT := 2;
    Temp : DINT := 0;
END_VAR

// Main Logic
IF N <= 2 THEN
    O := 1;
    F1 := 1;
    F2 := 1;
    Cnt := 2;
ELSE
    F1 := 1;
    F2 := 1;
    O := 1; // Default for N=1 or N=2, but N>2 so will be overwritten.
    Cnt := 2;

    WHILE (Cnt < N) DO
        // Calculate next Fibonacci number
        Temp := F1 + F2;

        // Apply saturation arithmetic: cap at 32767
        IF Temp > 32767 THEN
            Temp := 32767;
        END_IF;

        // Shift values for next iteration
        F1 := F2;
        F2 := Temp;

        // Update output and counter
        O := Temp;
        Cnt := Cnt + 1;

        // Exit loop if saturation limit reached
        IF Temp = 32767 THEN
            EXIT;
        END_IF;
    END_WHILE;
END_IF;

END_FUNCTION_BLOCK

(* ---- med_72.st ---- *)
FUNCTION_BLOCK DigitalSignageManagement
VAR_INPUT
    DisplayLocations : ARRAY[1..10] OF BOOL; (* TRUE = display active at location *)
    ContentSource : ARRAY[1..10] OF INT; (* Desired content: 1=News, 2=Weather, 3=Promo, 0/other=None *)
END_VAR

VAR_OUTPUT
    CurrentContent : ARRAY[1..10] OF INT; (* Actual displayed content: 1=News, 2=Weather, 3=Promo, 0=None *)
END_VAR

VAR
    i : INT; (* Loop counter *)
END_VAR

(* Main logic: Process all 10 locations each scan cycle *)
FOR i := 1 TO 10 DO
    IF DisplayLocations[i] THEN
        (* Display is active - validate and assign content *)
        CASE ContentSource[i] OF
            1: CurrentContent[i] := 1; (* News *)
            2: CurrentContent[i] := 2; (* Weather *)
            3: CurrentContent[i] := 3; (* Promotional Content *)
        ELSE
            CurrentContent[i] := 0; (* No Content for invalid code *)
        END_CASE;
    ELSE
        (* Display is inactive - force no content *)
        CurrentContent[i] := 0;
    END_IF;
END_FOR;

END_FUNCTION_BLOCK

(* ---- med_73.st ---- *)
FUNCTION_BLOCK RoboticWeldingSystem
VAR_INPUT
    RobotArm1Ready : BOOL;    (* Input for robot arm 1 ready status *)
    RobotArm2Ready : BOOL;    (* Input for robot arm 2 ready status *)
    WeldingGunReady : BOOL;   (* Input for welding gun ready status *)
    StartButton : BOOL;       (* Input for start button press *)
    StopButton : BOOL;        (* Input for stop button press *)
END_VAR

VAR_OUTPUT
    WeldingTrigger : BOOL;    (* Output to trigger welding *)
    WeldingComplete : BOOL;   (* Output indicating welding completion *)
END_VAR

VAR
    bAllReady : BOOL;         (* Internal flag for all components ready *)
    bStartCondition : BOOL;   (* Internal flag for valid start condition *)
END_VAR

(* Main logic for robotic welding system *)
(* Safety stop has highest priority - immediate stop when pressed *)
IF StopButton THEN
    WeldingTrigger := FALSE;
    WeldingComplete := TRUE;
ELSE
    (* Check if all components are ready *)
    bAllReady := RobotArm1Ready AND RobotArm2Ready AND WeldingGunReady;

    (* Check if start condition is met *)
    bStartCondition := bAllReady AND StartButton;

    (* Execute welding logic based on conditions *)
    IF bStartCondition THEN
        WeldingTrigger := TRUE;
        WeldingComplete := FALSE;
    ELSE
        WeldingTrigger := FALSE;
        WeldingComplete := TRUE;
    END_IF;
END_IF;

END_FUNCTION_BLOCK

(* ---- med_74.st ---- *)
(*
    TRAFFIC MANAGEMENT SYSTEM FUNCTION BLLOCK
    Description: Controls traffic lights for two independent road pairs based on vehicle counts.
    Logic: For each pair, the intersection with the higher vehicle count receives a green light (TRUE).
           In case of equal counts, a deterministic tie-breaker (alternating on equality) is applied.
           The system ensures exactly one green light per pair at all times.
    Design: Simple, deterministic, and robust with no external dependencies or timers.
*)

FUNCTION_BLOCK TrafficManagementSystem
VAR_INPUT
    VehicleCount1 : INT; (* Vehicle count at intersection 1 *)
    VehicleCount2 : INT; (* Vehicle count at intersection 2 *)
    VehicleCount3 : INT; (* Vehicle count at intersection 3 *)
    VehicleCount4 : INT; (* Vehicle count at intersection 4 *)
END_VAR
VAR_OUTPUT
    TrafficLight1 : BOOL; (* Green light control for intersection 1 *)
    TrafficLight2 : BOOL; (* Green light control for intersection 2 *)
    TrafficLight3 : BOOL; (* Green light control for intersection 3 *)
    TrafficLight4 : BOOL; (* Green light control for intersection 4 *)
END_VAR
VAR
    bPrevEqual1 : BOOL; (* Memory for tie-breaker state of pair 1 *)
    bPrevEqual2 : BOOL; (* Memory for tie-breaker state of pair 2 *)
END_VAR

(* Main execution logic *)
(* Process pair 1: Intersections 1 and 2 *)
IF VehicleCount1 > VehicleCount2 THEN
    TrafficLight1 := TRUE;
    TrafficLight2 := FALSE;
    bPrevEqual1 := FALSE; (* Reset tie-breaker memory on clear decision *)
ELSIF VehicleCount1 < VehicleCount2 THEN
    TrafficLight1 := FALSE;
    TrafficLight2 := TRUE;
    bPrevEqual1 := FALSE; (* Reset tie-breaker memory on clear decision *)
ELSE
    (* Equal counts: Apply deterministic tie-breaker (alternating) *)
    TrafficLight1 := NOT bPrevEqual1;
    TrafficLight2 := bPrevEqual1;
    bPrevEqual1 := NOT bPrevEqual1; (* Toggle state for next equality *)
END_IF;

(* Process pair 2: Intersections 3 and 4 *)
IF VehicleCount3 > VehicleCount4 THEN
    TrafficLight3 := TRUE;
    TrafficLight4 := FALSE;
    bPrevEqual2 := FALSE; (* Reset tie-breaker memory on clear decision *)
ELSIF VehicleCount3 < VehicleCount4 THEN
    TrafficLight3 := FALSE;
    TrafficLight4 := TRUE;
    bPrevEqual2 := FALSE; (* Reset tie-breaker memory on clear decision *)
ELSE
    (* Equal counts: Apply deterministic tie-breaker (alternating) *)
    TrafficLight3 := NOT bPrevEqual2;
    TrafficLight4 := bPrevEqual2;
    bPrevEqual2 := NOT bPrevEqual2; (* Toggle state for next equality *)
END_IF;

END_FUNCTION_BLOCK;
